LIN {X 0,Y 312.569,Z 301.55,A -85,B 0,C 180,E1 -15776.719,E2 -15776.719} C_VEL
LIN {X 0,Y 312.529,Z 301.553,A -85,B 0,C 180,E1 -15779.646,E2 -15779.646} C_VEL
LIN {X 0,Y 312.5,Z 301.556,A -85,B 0,C 180,E1 -15783.685,E2 -15783.685} C_VEL
LIN {X 0,Y 312.535,Z 301.555,A -85,B 0,C 180,E1 -15787.836,E2 -15787.836} C_VEL
LIN {X 0,Y 312.573,Z 301.686,A -85,B 0,C 180,E1 -15787.985,E2 -15787.985} C_VEL
LIN {X 0,Y 321.169,Z 326.946,A -85,B 0,C 180,E1 -15789.231,E2 -15789.231} C_VEL
LIN {X 0,Y 321.566,Z 328.599,A -85,B 0,C 180,E1 -15789.299,E2 -15789.299} C_VEL
LIN {X 0,Y 319.136,Z 408.879,A -85,B 0,C 180,E1 -15791.461,E2 -15791.461} C_VEL
LIN {X 0,Y 318.645,Z 421.58,A -85,B 0,C 180,E1 -15792.042,E2 -15792.042} C_VEL
LIN {X 0,Y 317.85,Z 434.866,A -85,B 0,C 180,E1 -15792.911,E2 -15792.911} C_VEL
LIN {X 0,Y 316.972,Z 446.153,A -85,B 0,C 180,E1 -15793.897,E2 -15793.897} C_VEL
LIN {X 0,Y 316.011,Z 457.09,A -85,B 0,C 180,E1 -15795.103,E2 -15795.103} C_VEL
LIN {X 0,Y 314.941,Z 468.05,A -85,B 0,C 180,E1 -15796.61,E2 -15796.61} C_VEL
LIN {X 0,Y 313.961,Z 477.57,A -85,B 0,C 180,E1 -15798.246,E2 -15798.246} C_VEL
LIN {X 0,Y 313.106,Z 485.746,A -85,B 0,C 180,E1 -15799.964,E2 -15799.964} C_VEL
LIN {X 0,Y 312.313,Z 493.408,A -85,B 0,C 180,E1 -15801.952,E2 -15801.952} C_VEL
LIN {X 0,Y 311.675,Z 499.881,A -85,B 0,C 180,E1 -15804.108,E2 -15804.108} C_VEL
LIN {X 0,Y 311.305,Z 504.728,A -85,B 0,C 180,E1 -15806.208,E2 -15806.208} C_VEL
LIN {X 0,Y 310.978,Z 507.716,A -85,B 0,C 180,E1 -15807.922,E2 -15807.922} C_VEL
LIN {X 0,Y 310.731,Z 510.421,A -85,B 0,C 180,E1 -15810.16,E2 -15810.16} C_VEL
LIN {X 0,Y 310.726,Z 511.311,A -85,B 0,C 180,E1 -15811.362,E2 -15811.362} C_VEL
LIN {X 0,Y 310.11,Z 511.982,A -85,B 0,C 180,E1 -15812.439,E2 -15812.439} C_VEL
LIN {X 0,Y 307.342,Z 512.482,A -85,B 0,C 180,E1 -15814.207,E2 -15814.207} C_VEL
LIN {X 0,Y 304.699,Z 512.119,A -85,B 0,C 180,E1 -15816.005,E2 -15816.005} C_VEL
LIN {X 0,Y 304.296,Z 511.437,A -85,B 0,C 180,E1 -15817.113,E2 -15817.113} C_VEL
LIN {X 0,Y 304.633,Z 510.361,A -85,B 0,C 180,E1 -15818.339,E2 -15818.339} C_VEL
LIN {X 0,Y 305.421,Z 507.392,A -85,B 0,C 180,E1 -15820.616,E2 -15820.616} C_VEL
LIN {X 0,Y 306.337,Z 503.587,A -85,B 0,C 180,E1 -15822.648,E2 -15822.648} C_VEL
LIN {X 0,Y 307.601,Z 498.313,A -85,B 0,C 180,E1 -15824.767,E2 -15824.767} C_VEL
LIN {X 0,Y 309.165,Z 491.514,A -85,B 0,C 180,E1 -15826.861,E2 -15826.861} C_VEL
LIN {X 0,Y 311.029,Z 482.961,A -85,B 0,C 180,E1 -15828.927,E2 -15828.927} C_VEL
LIN {X 0,Y 312.834,Z 473.936,A -85,B 0,C 180,E1 -15830.66,E2 -15830.66} C_VEL
LIN {X 0,Y 314.861,Z 463.188,A -85,B 0,C 180,E1 -15832.304,E2 -15832.304} C_VEL
LIN {X 0,Y 316.565,Z 452.402,A -85,B 0,C 180,E1 -15833.627,E2 -15833.627} C_VEL
LIN {X 0,Y 318.121,Z 440.675,A -85,B 0,C 180,E1 -15834.752,E2 -15834.752} C_VEL
LIN {X 0,Y 319.445,Z 428.246,A -85,B 0,C 180,E1 -15835.663,E2 -15835.663} C_VEL
LIN {X 0,Y 320.377,Z 416.205,A -85,B 0,C 180,E1 -15836.306,E2 -15836.306} C_VEL
LIN {X 0,Y 321.226,Z 399.512,A -85,B 0,C 180,E1 -15836.865,E2 -15836.865} C_VEL
LIN {X 0,Y 324.423,Z 337.687,A -85,B 0,C 180,E1 -15838.659,E2 -15838.659} C_VEL
LIN {X 0,Y 316.819,Z 321.614,A -85,B 0,C 180,E1 -15840.328,E2 -15840.328} C_VEL
LIN {X 0,Y 311.214,Z 311.88,A -85,B 0,C 180,E1 -15841.598,E2 -15841.598} C_VEL
LIN {X 0,Y 306.346,Z 304.341,A -85,B 0,C 180,E1 -15842.795,E2 -15842.795} C_VEL
LIN {X 0,Y 305.667,Z 302.413,A -85,B 0,C 180,E1 -15843.543,E2 -15843.543} C_VEL
LIN {X 0,Y 305.794,Z 302.393,A -85,B 0,C 180,E1 -15846.599,E2 -15846.599} C_VEL
LIN {X 0,Y 305.658,Z 302.414,A -85,B 0,C 180,E1 -15849.263,E2 -15849.263} C_VEL
LIN {X 0,Y 305.543,Z 302.423,A -85,B 0,C 180,E1 -15853.299,E2 -15853.299} C_VEL
LIN {X 0,Y 305.509,Z 302.428,A -85,B 0,C 180,E1 -15856.025,E2 -15856.025} C_VEL
LIN {X 0,Y 305.442,Z 302.43,A -85,B 0,C 180,E1 -15860.191,E2 -15860.191} C_VEL
LIN {X 0,Y 305.464,Z 302.435,A -85,B 0,C 180,E1 -15864.466,E2 -15864.466} C_VEL
LIN {X 0,Y 305.456,Z 302.438,A -85,B 0,C 180,E1 -15867.398,E2 -15867.398} C_VEL
LIN {X 0,Y 305.402,Z 302.443,A -85,B 0,C 180,E1 -15870.416,E2 -15870.416} C_VEL
LIN {X 0,Y 305.434,Z 302.433,A -85,B 0,C 180,E1 -15874.082,E2 -15874.082} C_VEL
LIN {X 0,Y 305.452,Z 302.432,A -85,B 0,C 180,E1 -15876.743,E2 -15876.743} C_VEL
LIN {X 0,Y 305.435,Z 302.434,A -85,B 0,C 180,E1 -15880.112,E2 -15880.112} C_VEL
LIN {X 0,Y 305.402,Z 302.443,A -85,B 0,C 180,E1 -15883.66,E2 -15883.66} C_VEL
LIN {X 0,Y 305.434,Z 302.44,A -85,B 0,C 180,E1 -15887.419,E2 -15887.419} C_VEL
LIN {X 0,Y 305.457,Z 302.437,A -85,B 0,C 180,E1 -15891.602,E2 -15891.602} C_VEL
LIN {X 0,Y 308.417,Z 311.804,A -85,B 0,C 180,E1 -15895.12,E2 -15895.12} C_VEL
LIN {X 0,Y 311.052,Z 321.561,A -85,B 0,C 180,E1 -15898.326,E2 -15898.326} C_VEL
LIN {X 0,Y 312.487,Z 328.352,A -85,B 0,C 180,E1 -15900.35,E2 -15900.35} C_VEL
LIN {X 0,Y 315.777,Z 336.016,A -85,B 0,C 180,E1 -15901.158,E2 -15901.158} C_VEL
LIN {X 0,Y 319.475,Z 354.495,A -85,B 0,C 180,E1 -15902.374,E2 -15902.374} C_VEL
LIN {X 0,Y 321.978,Z 372.44,A -85,B 0,C 180,E1 -15903.36,E2 -15903.36} C_VEL
LIN {X 0,Y 322.658,Z 381.327,A -85,B 0,C 180,E1 -15903.762,E2 -15903.762} C_VEL
LIN {X 0,Y 319.765,Z 440.74,A -85,B 0,C 180,E1 -15905.495,E2 -15905.495} C_VEL
LIN {X 0,Y 318.351,Z 455.279,A -85,B 0,C 180,E1 -15906.159,E2 -15906.159} C_VEL
LIN {X 0,Y 316.786,Z 467.665,A -85,B 0,C 180,E1 -15906.987,E2 -15906.987} C_VEL
LIN {X 0,Y 314.861,Z 479.761,A -85,B 0,C 180,E1 -15908.05,E2 -15908.05} C_VEL
LIN {X 0,Y 312.782,Z 491.982,A -85,B 0,C 180,E1 -15909.451,E2 -15909.451} C_VEL
LIN {X 0,Y 310.928,Z 501.887,A -85,B 0,C 180,E1 -15910.872,E2 -15910.872} C_VEL
LIN {X 0,Y 309.11,Z 510.986,A -85,B 0,C 180,E1 -15912.471,E2 -15912.471} C_VEL
LIN {X 0,Y 307.444,Z 519.938,A -85,B 0,C 180,E1 -15914.423,E2 -15914.423} C_VEL
LIN {X 0,Y 306.094,Z 527.138,A -85,B 0,C 180,E1 -15916.392,E2 -15916.392} C_VEL
LIN {X 0,Y 305.025,Z 532.101,A -85,B 0,C 180,E1 -15918.035,E2 -15918.035} C_VEL
LIN {X 0,Y 304.335,Z 536.915,A -85,B 0,C 180,E1 -15920.029,E2 -15920.029} C_VEL
LIN {X 0,Y 303.92,Z 540.631,A -85,B 0,C 180,E1 -15922.028,E2 -15922.028} C_VEL
LIN {X 0,Y 303.731,Z 543.552,A -85,B 0,C 180,E1 -15924.257,E2 -15924.257} C_VEL
LIN {X 0,Y 303.708,Z 545.024,A -85,B 0,C 180,E1 -15926.022,E2 -15926.022} C_VEL
LIN {X 0,Y 303.709,Z 545.634,A -85,B 0,C 180,E1 -15927.35,E2 -15927.35} C_VEL
LIN {X 0,Y 303.81,Z 545.808,A -85,B 0,C 180,E1 -15928.677,E2 -15928.677} C_VEL
LIN {X 0,Y 304.002,Z 545.577,A -85,B 0,C 180,E1 -15930.002,E2 -15930.002} C_VEL
LIN {X 0,Y 303.897,Z 544.913,A -85,B 0,C 180,E1 -15931.327,E2 -15931.327} C_VEL
LIN {X 0,Y 303.773,Z 543.775,A -85,B 0,C 180,E1 -15932.654,E2 -15932.654} C_VEL
LIN {X 0,Y 303.805,Z 541.247,A -85,B 0,C 180,E1 -15934.646,E2 -15934.646} C_VEL
LIN {X 0,Y 303.91,Z 537.616,A -85,B 0,C 180,E1 -15936.641,E2 -15936.641} C_VEL
LIN {X 0,Y 304.016,Z 532.776,A -85,B 0,C 180,E1 -15938.643,E2 -15938.643} C_VEL
LIN {X 0,Y 304.449,Z 526.612,A -85,B 0,C 180,E1 -15940.643,E2 -15940.643} C_VEL
LIN {X 0,Y 305.187,Z 518.907,A -85,B 0,C 180,E1 -15942.638,E2 -15942.638} C_VEL
LIN {X 0,Y 305.99,Z 511.012,A -85,B 0,C 180,E1 -15944.295,E2 -15944.295} C_VEL
LIN {X 0,Y 306.916,Z 501.329,A -85,B 0,C 180,E1 -15945.95,E2 -15945.95} C_VEL
LIN {X 0,Y 308.062,Z 490.632,A -85,B 0,C 180,E1 -15947.424,E2 -15947.424} C_VEL
LIN {X 0,Y 309.114,Z 480.385,A -85,B 0,C 180,E1 -15948.561,E2 -15948.561} C_VEL
LIN {X 0,Y 310.224,Z 468.373,A -85,B 0,C 180,E1 -15949.607,E2 -15949.607} C_VEL
LIN {X 0,Y 311.305,Z 454.669,A -85,B 0,C 180,E1 -15950.483,E2 -15950.483} C_VEL
LIN {X 0,Y 312.046,Z 441.896,A -85,B 0,C 180,E1 -15951.036,E2 -15951.036} C_VEL
LIN {X 0,Y 313.768,Z 376.823,A -85,B 0,C 180,E1 -15952.843,E2 -15952.843} C_VEL
LIN {X 0,Y 308.68,Z 334.134,A -85,B 0,C 180,E1 -15954.435,E2 -15954.435} C_VEL
LIN {X 0,Y 309.846,Z 324.126,A -85,B 0,C 180,E1 -15956.977,E2 -15956.977} C_VEL
LIN {X 0,Y 307.598,Z 312.592,A -85,B 0,C 180,E1 -15960.175,E2 -15960.175} C_VEL
LIN {X 0,Y 305.503,Z 302.431,A -85,B 0,C 180,E1 -15963.116,E2 -15963.116} C_VEL
LIN {X 0,Y 305.449,Z 302.439,A -85,B 0,C 180,E1 -15966.741,E2 -15966.741} C_VEL
LIN {X 0,Y 305.403,Z 302.443,A -85,B 0,C 180,E1 -15970.588,E2 -15970.588} C_VEL
LIN {X 0,Y 305.413,Z 302.438,A -85,B 0,C 180,E1 -15973.655,E2 -15973.655} C_VEL
LIN {X 0,Y 305.404,Z 302.44,A -85,B 0,C 180,E1 -15977.421,E2 -15977.421} C_VEL
LIN {X 0,Y 305.417,Z 302.438,A -85,B 0,C 180,E1 -15981.588,E2 -15981.588} C_VEL
LIN {X 0,Y 305.448,Z 302.438,A -85,B 0,C 180,E1 -15984.884,E2 -15984.884} C_VEL
LIN {X 0,Y 305.426,Z 302.437,A -85,B 0,C 180,E1 -15988.358,E2 -15988.358} C_VEL
LIN {X 0,Y 305.473,Z 302.436,A -85,B 0,C 180,E1 -15991.108,E2 -15991.108} C_VEL
LIN {X 0,Y 305.486,Z 302.429,A -85,B 0,C 180,E1 -15994.079,E2 -15994.079} C_VEL
LIN {X 0,Y 305.459,Z 302.436,A -85,B 0,C 180,E1 -15996.974,E2 -15996.974} C_VEL
LIN {X 0,Y 305.498,Z 302.433,A -85,B 0,C 180,E1 -16001.211,E2 -16001.211} C_VEL
LIN {X 0,Y 305.606,Z 302.419,A -85,B 0,C 180,E1 -16005.346,E2 -16005.346} C_VEL
LIN {X 0,Y 305.603,Z 302.42,A -85,B 0,C 180,E1 -16009.398,E2 -16009.398} C_VEL
LIN {X 0,Y 305.765,Z 302.395,A -85,B 0,C 180,E1 -16012.072,E2 -16012.072} C_VEL
LIN {X 0,Y 305.657,Z 302.408,A -85,B 0,C 180,E1 -16014.722,E2 -16014.722} C_VEL
LIN {X 0,Y 305.931,Z 302.374,A -85,B 0,C 180,E1 -16018.683,E2 -16018.683} C_VEL
LIN {X 0,Y 305.931,Z 302.378,A -85,B 0,C 180,E1 -16021.316,E2 -16021.316} C_VEL
LIN {X 0,Y 305.653,Z 302.411,A -85,B 0,C 180,E1 -16025.276,E2 -16025.276} C_VEL
LIN {X 0,Y 305.764,Z 302.397,A -85,B 0,C 180,E1 -16027.926,E2 -16027.926} C_VEL
LIN {X 0,Y 305.58,Z 302.42,A -85,B 0,C 180,E1 -16031.945,E2 -16031.945} C_VEL
LIN {X 0,Y 305.587,Z 302.417,A -85,B 0,C 180,E1 -16035.012,E2 -16035.012} C_VEL
LIN {X 0,Y 305.492,Z 302.428,A -85,B 0,C 180,E1 -16038.788,E2 -16038.788} C_VEL
LIN {X 0,Y 305.469,Z 302.432,A -85,B 0,C 180,E1 -16043.04,E2 -16043.04} C_VEL
LIN {X 0,Y 305.513,Z 302.427,A -85,B 0,C 180,E1 -16046.221,E2 -16046.221} C_VEL
LIN {X 0,Y 305.477,Z 302.43,A -85,B 0,C 180,E1 -16049.05,E2 -16049.05} C_VEL
LIN {X 0,Y 305.428,Z 302.441,A -85,B 0,C 180,E1 -16051.953,E2 -16051.953} C_VEL
LIN {X 0,Y 305.446,Z 302.434,A -85,B 0,C 180,E1 -16055.114,E2 -16055.114} C_VEL
LIN {X 0,Y 305.454,Z 302.434,A -85,B 0,C 180,E1 -16058.534,E2 -16058.534} C_VEL
LIN {X 0,Y 305.449,Z 302.434,A -85,B 0,C 180,E1 -16062.588,E2 -16062.588} C_VEL
LIN {X 0,Y 305.476,Z 302.433,A -85,B 0,C 180,E1 -16066.357,E2 -16066.357} C_VEL
LIN {X 0,Y 305.475,Z 302.434,A -85,B 0,C 180,E1 -16069.897,E2 -16069.897} C_VEL
LIN {X 0,Y 305.494,Z 302.429,A -85,B 0,C 180,E1 -16073.627,E2 -16073.627} C_VEL
LIN {X 0,Y 305.458,Z 302.436,A -85,B 0,C 180,E1 -16076.484,E2 -16076.484} C_VEL
LIN {X 0,Y 305.451,Z 302.434,A -85,B 0,C 180,E1 -16079.591,E2 -16079.591} C_VEL
LIN {X 0,Y 305.513,Z 302.428,A -85,B 0,C 180,E1 -16082.608,E2 -16082.608} C_VEL
LIN {X 0,Y 305.504,Z 302.427,A -85,B 0,C 180,E1 -16085.539,E2 -16085.539} C_VEL
LIN {X 0,Y 305.516,Z 302.426,A -85,B 0,C 180,E1 -16089.815,E2 -16089.815} C_VEL
LIN {X 0,Y 305.572,Z 302.422,A -85,B 0,C 180,E1 -16092.602,E2 -16092.602} C_VEL
LIN {X 0,Y 305.646,Z 302.409,A -85,B 0,C 180,E1 -16095.348,E2 -16095.348} C_VEL
LIN {X 0,Y 305.636,Z 302.41,A -85,B 0,C 180,E1 -16099.399,E2 -16099.399} C_VEL
LIN {X 0,Y 305.811,Z 302.39,A -85,B 0,C 180,E1 -16102.073,E2 -16102.073} C_VEL
LIN {X 0,Y 305.686,Z 302.408,A -85,B 0,C 180,E1 -16104.722,E2 -16104.722} C_VEL
LIN {X 0,Y 305.955,Z 302.376,A -85,B 0,C 180,E1 -16108.682,E2 -16108.682} C_VEL
LIN {X 0,Y 305.954,Z 302.371,A -85,B 0,C 180,E1 -16111.314,E2 -16111.314} C_VEL
LIN {X 0,Y 305.846,Z 302.388,A -85,B 0,C 180,E1 -16116.595,E2 -16116.595} C_VEL
LIN {X 0,Y 305.73,Z 302.4,A -85,B 0,C 180,E1 -16119.257,E2 -16119.257} C_VEL
LIN {X 0,Y 305.584,Z 302.419,A -85,B 0,C 180,E1 -16123.293,E2 -16123.293} C_VEL
LIN {X 0,Y 305.585,Z 302.416,A -85,B 0,C 180,E1 -16126.017,E2 -16126.017} C_VEL
LIN {X 0,Y 305.603,Z 302.416,A -85,B 0,C 180,E1 -16129.461,E2 -16129.461} C_VEL
LIN {X 0,Y 305.481,Z 302.435,A -85,B 0,C 180,E1 -16133.039,E2 -16133.039} C_VEL
LIN {X 0,Y 305.54,Z 302.423,A -85,B 0,C 180,E1 -16136.226,E2 -16136.226} C_VEL
LIN {X 0,Y 305.48,Z 302.436,A -85,B 0,C 180,E1 -16139.046,E2 -16139.046} C_VEL
LIN {X 0,Y 305.446,Z 302.436,A -85,B 0,C 180,E1 -16143.513,E2 -16143.513} C_VEL
LIN {X 0,Y 305.504,Z 302.431,A -85,B 0,C 180,E1 -16147.555,E2 -16147.555} C_VEL
LIN {X 0,Y 312.503,Z 322.639,A -85,B 0,C 180,E1 -16148.602,E2 -16148.602} C_VEL
LIN {X 0,Y 314.751,Z 329.425,A -85,B 0,C 180,E1 -16148.934,E2 -16148.934} C_VEL
LIN {X 0,Y 312.289,Z 408.997,A -85,B 0,C 180,E1 -16151.132,E2 -16151.132} C_VEL
LIN {X 0,Y 311.764,Z 421.741,A -85,B 0,C 180,E1 -16151.724,E2 -16151.724} C_VEL
LIN {X 0,Y 310.939,Z 435.162,A -85,B 0,C 180,E1 -16152.617,E2 -16152.617} C_VEL
LIN {X 0,Y 309.981,Z 447.296,A -85,B 0,C 180,E1 -16153.712,E2 -16153.712} C_VEL
LIN {X 0,Y 309,Z 457.772,A -85,B 0,C 180,E1 -16154.904,E2 -16154.904} C_VEL
LIN {X 0,Y 307.983,Z 468.06,A -85,B 0,C 180,E1 -16156.348,E2 -16156.348} C_VEL
LIN {X 0,Y 306.9,Z 478.402,A -85,B 0,C 180,E1 -16158.168,E2 -16158.168} C_VEL
LIN {X 0,Y 305.951,Z 486.707,A -85,B 0,C 180,E1 -16159.971,E2 -16159.971} C_VEL
LIN {X 0,Y 305.193,Z 494.139,A -85,B 0,C 180,E1 -16161.976,E2 -16161.976} C_VEL
LIN {X 0,Y 304.535,Z 500.825,A -85,B 0,C 180,E1 -16164.292,E2 -16164.292} C_VEL
LIN {X 0,Y 304.192,Z 505.321,A -85,B 0,C 180,E1 -16166.325,E2 -16166.325} C_VEL
LIN {X 0,Y 303.76,Z 509.324,A -85,B 0,C 180,E1 -16168.863,E2 -16168.863} C_VEL
LIN {X 0,Y 303.669,Z 511.812,A -85,B 0,C 180,E1 -16171.562,E2 -16171.562} C_VEL
LIN {X 0,Y 303.821,Z 512.519,A -85,B 0,C 180,E1 -16174.425,E2 -16174.425} C_VEL
LIN {X 0,Y 304.296,Z 511.437,A -85,B 0,C 180,E1 -16177.113,E2 -16177.113} C_VEL
LIN {X 0,Y 303.951,Z 510.564,A -85,B 0,C 180,E1 -16178.21,E2 -16178.21} C_VEL
LIN {X 0,Y 301.661,Z 508.799,A -85,B 0,C 180,E1 -16180.007,E2 -16180.007} C_VEL
LIN {X 0,Y 299.514,Z 506.398,A -85,B 0,C 180,E1 -16181.799,E2 -16181.799} C_VEL
LIN {X 0,Y 299.401,Z 504.432,A -85,B 0,C 180,E1 -16182.871,E2 -16182.871} C_VEL
LIN {X 0,Y 300.781,Z 499.083,A -85,B 0,C 180,E1 -16185.107,E2 -16185.107} C_VEL
LIN {X 0,Y 302.515,Z 492.13,A -85,B 0,C 180,E1 -16187.318,E2 -16187.318} C_VEL
LIN {X 0,Y 304.408,Z 483.974,A -85,B 0,C 180,E1 -16189.357,E2 -16189.357} C_VEL
LIN {X 0,Y 306.286,Z 475.271,A -85,B 0,C 180,E1 -16191.102,E2 -16191.102} C_VEL
LIN {X 0,Y 308.234,Z 465.715,A -85,B 0,C 180,E1 -16192.632,E2 -16192.632} C_VEL
LIN {X 0,Y 309.994,Z 455.269,A -85,B 0,C 180,E1 -16193.993,E2 -16193.993} C_VEL
LIN {X 0,Y 311.672,Z 444.087,A -85,B 0,C 180,E1 -16195.15,E2 -16195.15} C_VEL
LIN {X 0,Y 313.129,Z 431.723,A -85,B 0,C 180,E1 -16196.14,E2 -16196.14} C_VEL
LIN {X 0,Y 314.275,Z 419.181,A -85,B 0,C 180,E1 -16196.876,E2 -16196.876} C_VEL
LIN {X 0,Y 315.039,Z 406.996,A -85,B 0,C 180,E1 -16197.363,E2 -16197.363} C_VEL
LIN {X 0,Y 318.65,Z 339.96,A -85,B 0,C 180,E1 -16199.357,E2 -16199.357} C_VEL
LIN {X 0,Y 311.717,Z 325.283,A -85,B 0,C 180,E1 -16200.971,E2 -16200.971} C_VEL
LIN {X 0,Y 306.646,Z 316.358,A -85,B 0,C 180,E1 -16202.174,E2 -16202.174} C_VEL
LIN {X 0,Y 301.652,Z 308.919,A -85,B 0,C 180,E1 -16203.407,E2 -16203.407} C_VEL
LIN {X 0,Y 299.041,Z 305.144,A -85,B 0,C 180,E1 -16204.128,E2 -16204.128} C_VEL
LIN {X 0,Y 298.594,Z 303.291,A -85,B 0,C 180,E1 -16204.895,E2 -16204.895} C_VEL
LIN {X 0,Y 298.739,Z 303.273,A -85,B 0,C 180,E1 -16206.756,E2 -16206.756} C_VEL
LIN {X 0,Y 298.59,Z 303.293,A -85,B 0,C 180,E1 -16209.484,E2 -16209.484} C_VEL
LIN {X 0,Y 298.503,Z 303.303,A -85,B 0,C 180,E1 -16213.618,E2 -16213.618} C_VEL
LIN {X 0,Y 298.442,Z 303.31,A -85,B 0,C 180,E1 -16216.415,E2 -16216.415} C_VEL
LIN {X 0,Y 298.405,Z 303.31,A -85,B 0,C 180,E1 -16219.62,E2 -16219.62} C_VEL
LIN {X 0,Y 298.392,Z 303.311,A -85,B 0,C 180,E1 -16223.604,E2 -16223.604} C_VEL
LIN {X 0,Y 298.425,Z 303.307,A -85,B 0,C 180,E1 -16226.581,E2 -16226.581} C_VEL
LIN {X 0,Y 298.37,Z 303.316,A -85,B 0,C 180,E1 -16229.647,E2 -16229.647} C_VEL
LIN {X 0,Y 298.361,Z 303.318,A -85,B 0,C 180,E1 -16232.805,E2 -16232.805} C_VEL
LIN {X 0,Y 298.423,Z 303.307,A -85,B 0,C 180,E1 -16236.813,E2 -16236.813} C_VEL
LIN {X 0,Y 298.389,Z 303.312,A -85,B 0,C 180,E1 -16239.49,E2 -16239.49} C_VEL
LIN {X 0,Y 298.377,Z 303.317,A -85,B 0,C 180,E1 -16243.108,E2 -16243.108} C_VEL
LIN {X 0,Y 298.383,Z 303.315,A -85,B 0,C 180,E1 -16246.926,E2 -16246.926} C_VEL
LIN {X 0,Y 298.404,Z 303.446,A -85,B 0,C 180,E1 -16250.411,E2 -16250.411} C_VEL
LIN {X 0,Y 301.282,Z 312.125,A -85,B 0,C 180,E1 -16253.897,E2 -16253.897} C_VEL
LIN {X 0,Y 303.981,Z 321.75,A -85,B 0,C 180,E1 -16257.276,E2 -16257.276} C_VEL
LIN {X 0,Y 305.376,Z 327.791,A -85,B 0,C 180,E1 -16259.165,E2 -16259.165} C_VEL
LIN {X 0,Y 310.513,Z 339.127,A -85,B 0,C 180,E1 -16260.474,E2 -16260.474} C_VEL
LIN {X 0,Y 313.87,Z 356.502,A -85,B 0,C 180,E1 -16261.673,E2 -16261.673} C_VEL
LIN {X 0,Y 316.164,Z 373.165,A -85,B 0,C 180,E1 -16262.621,E2 -16262.621} C_VEL
LIN {X 0,Y 316.888,Z 381.023,A -85,B 0,C 180,E1 -16263.009,E2 -16263.009} C_VEL
LIN {X 0,Y 313.739,Z 440.814,A -85,B 0,C 180,E1 -16264.815,E2 -16264.815} C_VEL
LIN {X 0,Y 312.283,Z 455.163,A -85,B 0,C 180,E1 -16265.489,E2 -16265.489} C_VEL
LIN {X 0,Y 310.635,Z 467.444,A -85,B 0,C 180,E1 -16266.327,E2 -16266.327} C_VEL
LIN {X 0,Y 308.613,Z 479.502,A -85,B 0,C 180,E1 -16267.405,E2 -16267.405} C_VEL
LIN {X 0,Y 306.688,Z 490.483,A -85,B 0,C 180,E1 -16268.672,E2 -16268.672} C_VEL
LIN {X 0,Y 304.659,Z 500.524,A -85,B 0,C 180,E1 -16270.112,E2 -16270.112} C_VEL
LIN {X 0,Y 302.725,Z 509.719,A -85,B 0,C 180,E1 -16271.739,E2 -16271.739} C_VEL
LIN {X 0,Y 300.818,Z 518.805,A -85,B 0,C 180,E1 -16273.723,E2 -16273.723} C_VEL
LIN {X 0,Y 299.389,Z 526.169,A -85,B 0,C 180,E1 -16275.734,E2 -16275.734} C_VEL
LIN {X 0,Y 298.049,Z 532.096,A -85,B 0,C 180,E1 -16277.751,E2 -16277.751} C_VEL
LIN {X 0,Y 297.323,Z 536.809,A -85,B 0,C 180,E1 -16279.792,E2 -16279.792} C_VEL
LIN {X 0,Y 296.858,Z 540.427,A -85,B 0,C 180,E1 -16281.837,E2 -16281.837} C_VEL
LIN {X 0,Y 296.601,Z 543.687,A -85,B 0,C 180,E1 -16284.564,E2 -16284.564} C_VEL
LIN {X 0,Y 296.62,Z 544.695,A -85,B 0,C 180,E1 -16285.927,E2 -16285.927} C_VEL
LIN {X 0,Y 296.63,Z 545.239,A -85,B 0,C 180,E1 -16287.286,E2 -16287.286} C_VEL
LIN {X 0,Y 296.717,Z 545.375,A -85,B 0,C 180,E1 -16288.645,E2 -16288.645} C_VEL
LIN {X 0,Y 296.927,Z 545.108,A -85,B 0,C 180,E1 -16290.002,E2 -16290.002} C_VEL
LIN {X 0,Y 296.806,Z 544.383,A -85,B 0,C 180,E1 -16291.359,E2 -16291.359} C_VEL
LIN {X 0,Y 296.693,Z 543.183,A -85,B 0,C 180,E1 -16292.717,E2 -16292.717} C_VEL
LIN {X 0,Y 296.732,Z 540.567,A -85,B 0,C 180,E1 -16294.757,E2 -16294.757} C_VEL
LIN {X 0,Y 296.84,Z 536.847,A -85,B 0,C 180,E1 -16296.8,E2 -16296.8} C_VEL
LIN {X 0,Y 296.965,Z 531.91,A -85,B 0,C 180,E1 -16298.85,E2 -16298.85} C_VEL
LIN {X 0,Y 297.42,Z 525.64,A -85,B 0,C 180,E1 -16300.898,E2 -16300.898} C_VEL
LIN {X 0,Y 298.193,Z 517.798,A -85,B 0,C 180,E1 -16302.939,E2 -16302.939} C_VEL
LIN {X 0,Y 299.084,Z 509.731,A -85,B 0,C 180,E1 -16304.633,E2 -16304.633} C_VEL
LIN {X 0,Y 300.055,Z 499.854,A -85,B 0,C 180,E1 -16306.325,E2 -16306.325} C_VEL
LIN {X 0,Y 301.271,Z 488.949,A -85,B 0,C 180,E1 -16307.829,E2 -16307.829} C_VEL
LIN {X 0,Y 302.563,Z 476.631,A -85,B 0,C 180,E1 -16309.154,E2 -16309.154} C_VEL
LIN {X 0,Y 303.669,Z 464.764,A -85,B 0,C 180,E1 -16310.137,E2 -16310.137} C_VEL
LIN {X 0,Y 304.563,Z 452.075,A -85,B 0,C 180,E1 -16310.913,E2 -16310.913} C_VEL
LIN {X 0,Y 305.266,Z 439.188,A -85,B 0,C 180,E1 -16311.437,E2 -16311.437} C_VEL
LIN {X 0,Y 306.954,Z 377.521,A -85,B 0,C 180,E1 -16313.197,E2 -16313.197} C_VEL
LIN {X 0,Y 301.816,Z 333.82,A -85,B 0,C 180,E1 -16314.854,E2 -16314.854} C_VEL
LIN {X 0,Y 302.819,Z 325.9,A -85,B 0,C 180,E1 -16316.908,E2 -16316.908} C_VEL
LIN {X 0,Y 301.341,Z 317.262,A -85,B 0,C 180,E1 -16319.325,E2 -16319.325} C_VEL
LIN {X 0,Y 298.446,Z 303.309,A -85,B 0,C 180,E1 -16323.422,E2 -16323.422} C_VEL
LIN {X 0,Y 298.385,Z 303.313,A -85,B 0,C 180,E1 -16327.761,E2 -16327.761} C_VEL
LIN {X 0,Y 298.341,Z 303.321,A -85,B 0,C 180,E1 -16331.267,E2 -16331.267} C_VEL
LIN {X 0,Y 298.349,Z 303.322,A -85,B 0,C 180,E1 -16335.033,E2 -16335.033} C_VEL
LIN {X 0,Y 298.332,Z 303.326,A -85,B 0,C 180,E1 -16338.921,E2 -16338.921} C_VEL
LIN {X 0,Y 298.367,Z 303.316,A -85,B 0,C 180,E1 -16342.234,E2 -16342.234} C_VEL
LIN {X 0,Y 298.395,Z 303.314,A -85,B 0,C 180,E1 -16345.579,E2 -16345.579} C_VEL
LIN {X 0,Y 298.362,Z 303.32,A -85,B 0,C 180,E1 -16348.787,E2 -16348.787} C_VEL
LIN {X 0,Y 298.409,Z 303.311,A -85,B 0,C 180,E1 -16351.898,E2 -16351.898} C_VEL
LIN {X 0,Y 298.424,Z 303.312,A -85,B 0,C 180,E1 -16354.918,E2 -16354.918} C_VEL
LIN {X 0,Y 298.382,Z 303.314,A -85,B 0,C 180,E1 -16357.86,E2 -16357.86} C_VEL
LIN {X 0,Y 298.445,Z 303.308,A -85,B 0,C 180,E1 -16360.75,E2 -16360.75} C_VEL
LIN {X 0,Y 298.57,Z 303.293,A -85,B 0,C 180,E1 -16364.993,E2 -16364.993} C_VEL
LIN {X 0,Y 298.562,Z 303.295,A -85,B 0,C 180,E1 -16369.145,E2 -16369.145} C_VEL
LIN {X 0,Y 298.711,Z 303.274,A -85,B 0,C 180,E1 -16371.884,E2 -16371.884} C_VEL
LIN {X 0,Y 298.628,Z 303.283,A -85,B 0,C 180,E1 -16374.598,E2 -16374.598} C_VEL
LIN {X 0,Y 298.898,Z 303.25,A -85,B 0,C 180,E1 -16378.652,E2 -16378.652} C_VEL
LIN {X 0,Y 298.897,Z 303.254,A -85,B 0,C 180,E1 -16381.347,E2 -16381.347} C_VEL
LIN {X 0,Y 298.75,Z 303.268,A -85,B 0,C 180,E1 -16386.754,E2 -16386.754} C_VEL
LIN {X 0,Y 298.611,Z 303.29,A -85,B 0,C 180,E1 -16389.482,E2 -16389.482} C_VEL
LIN {X 0,Y 298.522,Z 303.302,A -85,B 0,C 180,E1 -16393.616,E2 -16393.616} C_VEL
LIN {X 0,Y 298.458,Z 303.305,A -85,B 0,C 180,E1 -16396.413,E2 -16396.413} C_VEL
LIN {X 0,Y 298.423,Z 303.313,A -85,B 0,C 180,E1 -16399.617,E2 -16399.617} C_VEL
LIN {X 0,Y 298.411,Z 303.314,A -85,B 0,C 180,E1 -16403.601,E2 -16403.601} C_VEL
LIN {X 0,Y 298.471,Z 303.303,A -85,B 0,C 180,E1 -16406.575,E2 -16406.575} C_VEL
LIN {X 0,Y 298.404,Z 303.315,A -85,B 0,C 180,E1 -16409.642,E2 -16409.642} C_VEL
LIN {X 0,Y 298.38,Z 303.314,A -85,B 0,C 180,E1 -16412.801,E2 -16412.801} C_VEL
LIN {X 0,Y 298.432,Z 303.307,A -85,B 0,C 180,E1 -16416.808,E2 -16416.808} C_VEL
LIN {X 0,Y 298.397,Z 303.314,A -85,B 0,C 180,E1 -16419.487,E2 -16419.487} C_VEL
LIN {X 0,Y 298.388,Z 303.313,A -85,B 0,C 180,E1 -16423.104,E2 -16423.104} C_VEL
LIN {X 0,Y 298.429,Z 303.308,A -85,B 0,C 180,E1 -16426.928,E2 -16426.928} C_VEL
LIN {X 0,Y 298.421,Z 303.311,A -85,B 0,C 180,E1 -16430.518,E2 -16430.518} C_VEL
LIN {X 0,Y 298.426,Z 303.311,A -85,B 0,C 180,E1 -16433.933,E2 -16433.933} C_VEL
LIN {X 0,Y 298.387,Z 303.317,A -85,B 0,C 180,E1 -16437.985,E2 -16437.985} C_VEL
LIN {X 0,Y 298.453,Z 303.307,A -85,B 0,C 180,E1 -16441.904,E2 -16441.904} C_VEL
LIN {X 0,Y 298.481,Z 303.303,A -85,B 0,C 180,E1 -16444.924,E2 -16444.924} C_VEL
LIN {X 0,Y 298.455,Z 303.304,A -85,B 0,C 180,E1 -16449.316,E2 -16449.316} C_VEL
LIN {X 0,Y 298.535,Z 303.298,A -85,B 0,C 180,E1 -16452.179,E2 -16452.179} C_VEL
LIN {X 0,Y 298.591,Z 303.289,A -85,B 0,C 180,E1 -16454.994,E2 -16454.994} C_VEL
LIN {X 0,Y 298.591,Z 303.288,A -85,B 0,C 180,E1 -16459.145,E2 -16459.145} C_VEL
LIN {X 0,Y 298.756,Z 303.268,A -85,B 0,C 180,E1 -16461.885,E2 -16461.885} C_VEL
LIN {X 0,Y 298.658,Z 303.285,A -85,B 0,C 180,E1 -16464.597,E2 -16464.597} C_VEL
LIN {X 0,Y 298.921,Z 303.252,A -85,B 0,C 180,E1 -16468.651,E2 -16468.651} C_VEL
LIN {X 0,Y 298.921,Z 303.247,A -85,B 0,C 180,E1 -16471.345,E2 -16471.345} C_VEL
LIN {X 0,Y 298.792,Z 303.269,A -85,B 0,C 180,E1 -16476.751,E2 -16476.751} C_VEL
LIN {X 0,Y 298.675,Z 303.278,A -85,B 0,C 180,E1 -16479.477,E2 -16479.477} C_VEL
LIN {X 0,Y 298.546,Z 303.294,A -85,B 0,C 180,E1 -16483.612,E2 -16483.612} C_VEL
LIN {X 0,Y 298.541,Z 303.296,A -85,B 0,C 180,E1 -16486.405,E2 -16486.405} C_VEL
LIN {X 0,Y 298.532,Z 303.296,A -85,B 0,C 180,E1 -16489.667,E2 -16489.667} C_VEL
LIN {X 0,Y 298.447,Z 303.307,A -85,B 0,C 180,E1 -16493.594,E2 -16493.594} C_VEL
LIN {X 0,Y 298.478,Z 303.304,A -85,B 0,C 180,E1 -16496.57,E2 -16496.57} C_VEL
LIN {X 0,Y 298.405,Z 303.312,A -85,B 0,C 180,E1 -16499.637,E2 -16499.637} C_VEL
LIN {X 0,Y 298.377,Z 303.318,A -85,B 0,C 180,E1 -16502.796,E2 -16502.796} C_VEL
LIN {X 0,Y 298.446,Z 303.311,A -85,B 0,C 180,E1 -16506.927,E2 -16506.927} C_VEL
LIN {X 0,Y 298.439,Z 303.312,A -85,B 0,C 180,E1 -16507.145,E2 -16507.145} C_VEL
LIN {X 0,Y 305.918,Z 324.639,A -85,B 0,C 180,E1 -16508.277,E2 -16508.277} C_VEL
LIN {X 0,Y 307.933,Z 330.728,A -85,B 0,C 180,E1 -16508.579,E2 -16508.579} C_VEL
LIN {X 0,Y 305.415,Z 409.265,A -85,B 0,C 180,E1 -16510.814,E2 -16510.814} C_VEL
LIN {X 0,Y 304.877,Z 422.037,A -85,B 0,C 180,E1 -16511.421,E2 -16511.421} C_VEL
LIN {X 0,Y 304.067,Z 435.063,A -85,B 0,C 180,E1 -16512.302,E2 -16512.302} C_VEL
LIN {X 0,Y 303.138,Z 446.464,A -85,B 0,C 180,E1 -16513.332,E2 -16513.332} C_VEL
LIN {X 0,Y 301.939,Z 458.909,A -85,B 0,C 180,E1 -16514.772,E2 -16514.772} C_VEL
LIN {X 0,Y 300.87,Z 469.844,A -85,B 0,C 180,E1 -16516.387,E2 -16516.387} C_VEL
LIN {X 0,Y 299.76,Z 479.778,A -85,B 0,C 180,E1 -16518.211,E2 -16518.211} C_VEL
LIN {X 0,Y 298.786,Z 488.221,A -85,B 0,C 180,E1 -16520.137,E2 -16520.137} C_VEL
LIN {X 0,Y 298.033,Z 495.399,A -85,B 0,C 180,E1 -16522.186,E2 -16522.186} C_VEL
LIN {X 0,Y 297.477,Z 501.079,A -85,B 0,C 180,E1 -16524.217,E2 -16524.217} C_VEL
LIN {X 0,Y 297.071,Z 505.893,A -85,B 0,C 180,E1 -16526.439,E2 -16526.439} C_VEL
LIN {X 0,Y 296.697,Z 509.305,A -85,B 0,C 180,E1 -16528.593,E2 -16528.593} C_VEL
LIN {X 0,Y 296.573,Z 511.914,A -85,B 0,C 180,E1 -16531.244,E2 -16531.244} C_VEL
LIN {X 0,Y 296.591,Z 512.84,A -85,B 0,C 180,E1 -16533.243,E2 -16533.243} C_VEL
LIN {X 0,Y 296.788,Z 512.939,A -85,B 0,C 180,E1 -16534.771,E2 -16534.771} C_VEL
LIN {X 0,Y 297.241,Z 512.014,A -85,B 0,C 180,E1 -16537.219,E2 -16537.219} C_VEL
LIN {X 0,Y 297.875,Z 510.167,A -85,B 0,C 180,E1 -16539.274,E2 -16539.274} C_VEL
LIN {X 0,Y 298.714,Z 507.058,A -85,B 0,C 180,E1 -16541.482,E2 -16541.482} C_VEL
LIN {X 0,Y 299.401,Z 504.432,A -85,B 0,C 180,E1 -16542.871,E2 -16542.871} C_VEL
LIN {X 0,Y 299.374,Z 502.291,A -85,B 0,C 180,E1 -16543.924,E2 -16543.924} C_VEL
LIN {X 0,Y 297.704,Z 498.521,A -85,B 0,C 180,E1 -16545.655,E2 -16545.655} C_VEL
LIN {X 0,Y 296.163,Z 494.144,A -85,B 0,C 180,E1 -16547.344,E2 -16547.344} C_VEL
LIN {X 0,Y 296.331,Z 491.002,A -85,B 0,C 180,E1 -16548.313,E2 -16548.313} C_VEL
LIN {X 0,Y 298.181,Z 483.485,A -85,B 0,C 180,E1 -16550.162,E2 -16550.162} C_VEL
LIN {X 0,Y 300.213,Z 474.543,A -85,B 0,C 180,E1 -16551.926,E2 -16551.926} C_VEL
LIN {X 0,Y 302.567,Z 463.247,A -85,B 0,C 180,E1 -16553.7,E2 -16553.7} C_VEL
LIN {X 0,Y 304.416,Z 452.575,A -85,B 0,C 180,E1 -16555.034,E2 -16555.034} C_VEL
LIN {X 0,Y 306.329,Z 439.52,A -85,B 0,C 180,E1 -16556.301,E2 -16556.301} C_VEL
LIN {X 0,Y 307.8,Z 426.69,A -85,B 0,C 180,E1 -16557.22,E2 -16557.22} C_VEL
LIN {X 0,Y 308.839,Z 413.612,A -85,B 0,C 180,E1 -16557.885,E2 -16557.885} C_VEL
LIN {X 0,Y 312.958,Z 342.452,A -85,B 0,C 180,E1 -16560.084,E2 -16560.084} C_VEL
LIN {X 0,Y 307.145,Z 329.862,A -85,B 0,C 180,E1 -16561.515,E2 -16561.515} C_VEL
LIN {X 0,Y 302.402,Z 321.304,A -85,B 0,C 180,E1 -16562.715,E2 -16562.715} C_VEL
LIN {X 0,Y 297.658,Z 314.108,A -85,B 0,C 180,E1 -16563.935,E2 -16563.935} C_VEL
LIN {X 0,Y 292.067,Z 306.004,A -85,B 0,C 180,E1 -16565.524,E2 -16565.524} C_VEL
LIN {X 0,Y 291.666,Z 304.153,A -85,B 0,C 180,E1 -16566.399,E2 -16566.399} C_VEL
LIN {X 0,Y 291.532,Z 304.17,A -85,B 0,C 180,E1 -16569.716,E2 -16569.716} C_VEL
LIN {X 0,Y 291.474,Z 304.179,A -85,B 0,C 180,E1 -16573.953,E2 -16573.953} C_VEL
LIN {X 0,Y 291.387,Z 304.186,A -85,B 0,C 180,E1 -16576.824,E2 -16576.824} C_VEL
LIN {X 0,Y 291.355,Z 304.186,A -85,B 0,C 180,E1 -16579.845,E2 -16579.845} C_VEL
LIN {X 0,Y 291.343,Z 304.193,A -85,B 0,C 180,E1 -16584.211,E2 -16584.211} C_VEL
LIN {X 0,Y 291.368,Z 304.192,A -85,B 0,C 180,E1 -16587.278,E2 -16587.278} C_VEL
LIN {X 0,Y 291.29,Z 304.202,A -85,B 0,C 180,E1 -16590.443,E2 -16590.443} C_VEL
LIN {X 0,Y 291.313,Z 304.194,A -85,B 0,C 180,E1 -16593.703,E2 -16593.703} C_VEL
LIN {X 0,Y 291.36,Z 304.186,A -85,B 0,C 180,E1 -16597.261,E2 -16597.261} C_VEL
LIN {X 0,Y 291.313,Z 304.197,A -85,B 0,C 180,E1 -16600.647,E2 -16600.647} C_VEL
LIN {X 0,Y 291.269,Z 304.2,A -85,B 0,C 180,E1 -16604.407,E2 -16604.407} C_VEL
LIN {X 0,Y 291.309,Z 304.197,A -85,B 0,C 180,E1 -16608.59,E2 -16608.59} C_VEL
LIN {X 0,Y 291.357,Z 304.341,A -85,B 0,C 180,E1 -16608.985,E2 -16608.985} C_VEL
LIN {X 0,Y 293.774,Z 311.494,A -85,B 0,C 180,E1 -16612.136,E2 -16612.136} C_VEL
LIN {X 0,Y 295.992,Z 318.576,A -85,B 0,C 180,E1 -16614.914,E2 -16614.914} C_VEL
LIN {X 0,Y 298.169,Z 326.91,A -85,B 0,C 180,E1 -16617.823,E2 -16617.823} C_VEL
LIN {X 0,Y 303.773,Z 338.761,A -85,B 0,C 180,E1 -16619.364,E2 -16619.364} C_VEL
LIN {X 0,Y 305.611,Z 343.284,A -85,B 0,C 180,E1 -16619.862,E2 -16619.862} C_VEL
LIN {X 0,Y 308.841,Z 361.489,A -85,B 0,C 180,E1 -16621.122,E2 -16621.122} C_VEL
LIN {X 0,Y 310.887,Z 378.75,A -85,B 0,C 180,E1 -16622.107,E2 -16622.107} C_VEL
LIN {X 0,Y 311.076,Z 383.685,A -85,B 0,C 180,E1 -16622.323,E2 -16622.323} C_VEL
LIN {X 0,Y 307.95,Z 439.704,A -85,B 0,C 180,E1 -16624.04,E2 -16624.04} C_VEL
LIN {X 0,Y 306.473,Z 454.008,A -85,B 0,C 180,E1 -16624.721,E2 -16624.721} C_VEL
LIN {X 0,Y 304.849,Z 465.454,A -85,B 0,C 180,E1 -16625.487,E2 -16625.487} C_VEL
LIN {X 0,Y 302.721,Z 477.723,A -85,B 0,C 180,E1 -16626.578,E2 -16626.578} C_VEL
LIN {X 0,Y 300.372,Z 490.193,A -85,B 0,C 180,E1 -16628.02,E2 -16628.02} C_VEL
LIN {X 0,Y 298.033,Z 501.195,A -85,B 0,C 180,E1 -16629.65,E2 -16629.65} C_VEL
LIN {X 0,Y 296.005,Z 510.224,A -85,B 0,C 180,E1 -16631.309,E2 -16631.309} C_VEL
LIN {X 0,Y 294.015,Z 519.114,A -85,B 0,C 180,E1 -16633.335,E2 -16633.335} C_VEL
LIN {X 0,Y 292.503,Z 526.273,A -85,B 0,C 180,E1 -16635.391,E2 -16635.391} C_VEL
LIN {X 0,Y 291.088,Z 532.092,A -85,B 0,C 180,E1 -16637.453,E2 -16637.453} C_VEL
LIN {X 0,Y 290.303,Z 536.713,A -85,B 0,C 180,E1 -16639.542,E2 -16639.542} C_VEL
LIN {X 0,Y 289.816,Z 540.245,A -85,B 0,C 180,E1 -16641.637,E2 -16641.637} C_VEL
LIN {X 0,Y 289.537,Z 543.418,A -85,B 0,C 180,E1 -16644.431,E2 -16644.431} C_VEL
LIN {X 0,Y 289.534,Z 544.343,A -85,B 0,C 180,E1 -16645.827,E2 -16645.827} C_VEL
LIN {X 0,Y 289.552,Z 544.847,A -85,B 0,C 180,E1 -16647.22,E2 -16647.22} C_VEL
LIN {X 0,Y 289.624,Z 544.945,A -85,B 0,C 180,E1 -16648.612,E2 -16648.612} C_VEL
LIN {X 0,Y 289.838,Z 544.636,A -85,B 0,C 180,E1 -16650.002,E2 -16650.002} C_VEL
LIN {X 0,Y 289.715,Z 543.833,A -85,B 0,C 180,E1 -16651.392,E2 -16651.392} C_VEL
LIN {X 0,Y 289.617,Z 542.592,A -85,B 0,C 180,E1 -16652.784,E2 -16652.784} C_VEL
LIN {X 0,Y 289.664,Z 539.887,A -85,B 0,C 180,E1 -16654.873,E2 -16654.873} C_VEL
LIN {X 0,Y 289.749,Z 536.068,A -85,B 0,C 180,E1 -16656.967,E2 -16656.967} C_VEL
LIN {X 0,Y 289.925,Z 531.029,A -85,B 0,C 180,E1 -16659.067,E2 -16659.067} C_VEL
LIN {X 0,Y 290.376,Z 524.635,A -85,B 0,C 180,E1 -16661.166,E2 -16661.166} C_VEL
LIN {X 0,Y 291.228,Z 516.601,A -85,B 0,C 180,E1 -16663.254,E2 -16663.254} C_VEL
LIN {X 0,Y 292.176,Z 508.372,A -85,B 0,C 180,E1 -16664.987,E2 -16664.987} C_VEL
LIN {X 0,Y 293.026,Z 499.739,A -85,B 0,C 180,E1 -16666.49,E2 -16666.49} C_VEL
LIN {X 0,Y 294.131,Z 489.761,A -85,B 0,C 180,E1 -16667.917,E2 -16667.917} C_VEL
LIN {X 0,Y 295.205,Z 479.495,A -85,B 0,C 180,E1 -16669.108,E2 -16669.108} C_VEL
LIN {X 0,Y 296.405,Z 467.475,A -85,B 0,C 180,E1 -16670.2,E2 -16670.2} C_VEL
LIN {X 0,Y 297.55,Z 453.804,A -85,B 0,C 180,E1 -16671.112,E2 -16671.112} C_VEL
LIN {X 0,Y 298.31,Z 441.055,A -85,B 0,C 180,E1 -16671.69,E2 -16671.69} C_VEL
LIN {X 0,Y 300.103,Z 378.168,A -85,B 0,C 180,E1 -16673.54,E2 -16673.54} C_VEL
LIN {X 0,Y 294.914,Z 333.524,A -85,B 0,C 180,E1 -16675.272,E2 -16675.272} C_VEL
LIN {X 0,Y 295.762,Z 326.218,A -85,B 0,C 180,E1 -16677.221,E2 -16677.221} C_VEL
LIN {X 0,Y 293.867,Z 316.115,A -85,B 0,C 180,E1 -16680.147,E2 -16680.147} C_VEL
LIN {X 0,Y 291.392,Z 304.188,A -85,B 0,C 180,E1 -16683.791,E2 -16683.791} C_VEL
LIN {X 0,Y 291.35,Z 304.191,A -85,B 0,C 180,E1 -16687.246,E2 -16687.246} C_VEL
LIN {X 0,Y 291.288,Z 304.198,A -85,B 0,C 180,E1 -16691.586,E2 -16691.586} C_VEL
LIN {X 0,Y 291.274,Z 304.199,A -85,B 0,C 180,E1 -16695.594,E2 -16695.594} C_VEL
LIN {X 0,Y 291.286,Z 304.2,A -85,B 0,C 180,E1 -16699.349,E2 -16699.349} C_VEL
LIN {X 0,Y 291.371,Z 304.192,A -85,B 0,C 180,E1 -16702.913,E2 -16702.913} C_VEL
LIN {X 0,Y 291.33,Z 304.193,A -85,B 0,C 180,E1 -16706.299,E2 -16706.299} C_VEL
LIN {X 0,Y 291.356,Z 304.19,A -85,B 0,C 180,E1 -16710.265,E2 -16710.265} C_VEL
LIN {X 0,Y 291.345,Z 304.191,A -85,B 0,C 180,E1 -16714.264,E2 -16714.264} C_VEL
LIN {X 0,Y 291.347,Z 304.194,A -85,B 0,C 180,E1 -16717.296,E2 -16717.296} C_VEL
LIN {X 0,Y 291.373,Z 304.187,A -85,B 0,C 180,E1 -16720.263,E2 -16720.263} C_VEL
LIN {X 0,Y 291.481,Z 304.174,A -85,B 0,C 180,E1 -16724.664,E2 -16724.664} C_VEL
LIN {X 0,Y 291.508,Z 304.172,A -85,B 0,C 180,E1 -16728.879,E2 -16728.879} C_VEL
LIN {X 0,Y 291.659,Z 304.154,A -85,B 0,C 180,E1 -16731.686,E2 -16731.686} C_VEL
LIN {X 0,Y 291.599,Z 304.158,A -85,B 0,C 180,E1 -16734.467,E2 -16734.467} C_VEL
LIN {X 0,Y 291.864,Z 304.126,A -85,B 0,C 180,E1 -16738.62,E2 -16738.62} C_VEL
LIN {X 0,Y 291.864,Z 304.13,A -85,B 0,C 180,E1 -16741.379,E2 -16741.379} C_VEL
LIN {X 0,Y 291.7,Z 304.147,A -85,B 0,C 180,E1 -16746.918,E2 -16746.918} C_VEL
LIN {X 0,Y 291.553,Z 304.168,A -85,B 0,C 180,E1 -16749.714,E2 -16749.714} C_VEL
LIN {X 0,Y 291.494,Z 304.175,A -85,B 0,C 180,E1 -16753.951,E2 -16753.951} C_VEL
LIN {X 0,Y 291.403,Z 304.183,A -85,B 0,C 180,E1 -16756.822,E2 -16756.822} C_VEL
LIN {X 0,Y 291.374,Z 304.191,A -85,B 0,C 180,E1 -16759.842,E2 -16759.842} C_VEL
LIN {X 0,Y 291.365,Z 304.19,A -85,B 0,C 180,E1 -16764.208,E2 -16764.208} C_VEL
LIN {X 0,Y 291.405,Z 304.184,A -85,B 0,C 180,E1 -16767.272,E2 -16767.272} C_VEL
LIN {X 0,Y 291.321,Z 304.195,A -85,B 0,C 180,E1 -16770.438,E2 -16770.438} C_VEL
LIN {X 0,Y 291.329,Z 304.196,A -85,B 0,C 180,E1 -16773.699,E2 -16773.699} C_VEL
LIN {X 0,Y 291.367,Z 304.188,A -85,B 0,C 180,E1 -16777.256,E2 -16777.256} C_VEL
LIN {X 0,Y 291.326,Z 304.194,A -85,B 0,C 180,E1 -16780.643,E2 -16780.643} C_VEL
LIN {X 0,Y 291.305,Z 304.197,A -85,B 0,C 180,E1 -16784.398,E2 -16784.398} C_VEL
LIN {X 0,Y 291.371,Z 304.19,A -85,B 0,C 180,E1 -16788.393,E2 -16788.393} C_VEL
LIN {X 0,Y 291.376,Z 304.186,A -85,B 0,C 180,E1 -16791.164,E2 -16791.164} C_VEL
LIN {X 0,Y 291.379,Z 304.188,A -85,B 0,C 180,E1 -16794.63,E2 -16794.63} C_VEL
LIN {X 0,Y 291.364,Z 304.191,A -85,B 0,C 180,E1 -16797.951,E2 -16797.951} C_VEL
LIN {X 0,Y 291.372,Z 304.186,A -85,B 0,C 180,E1 -16801.158,E2 -16801.158} C_VEL
LIN {X 0,Y 291.411,Z 304.188,A -85,B 0,C 180,E1 -16804.272,E2 -16804.272} C_VEL
LIN {X 0,Y 291.385,Z 304.185,A -85,B 0,C 180,E1 -16807.3,E2 -16807.3} C_VEL
LIN {X 0,Y 291.456,Z 304.18,A -85,B 0,C 180,E1 -16810.27,E2 -16810.27} C_VEL
LIN {X 0,Y 291.553,Z 304.168,A -85,B 0,C 180,E1 -16814.623,E2 -16814.623} C_VEL
LIN {X 0,Y 291.535,Z 304.169,A -85,B 0,C 180,E1 -16818.879,E2 -16818.879} C_VEL
LIN {X 0,Y 291.707,Z 304.146,A -85,B 0,C 180,E1 -16821.687,E2 -16821.687} C_VEL
LIN {X 0,Y 291.628,Z 304.16,A -85,B 0,C 180,E1 -16824.467,E2 -16824.467} C_VEL
LIN {X 0,Y 291.887,Z 304.128,A -85,B 0,C 180,E1 -16828.618,E2 -16828.618} C_VEL
LIN {X 0,Y 291.887,Z 304.124,A -85,B 0,C 180,E1 -16831.377,E2 -16831.377} C_VEL
LIN {X 0,Y 291.741,Z 304.145,A -85,B 0,C 180,E1 -16836.915,E2 -16836.915} C_VEL
LIN {X 0,Y 291.624,Z 304.156,A -85,B 0,C 180,E1 -16839.709,E2 -16839.709} C_VEL
LIN {X 0,Y 291.516,Z 304.17,A -85,B 0,C 180,E1 -16843.947,E2 -16843.947} C_VEL
LIN {X 0,Y 291.48,Z 304.178,A -85,B 0,C 180,E1 -16846.814,E2 -16846.814} C_VEL
LIN {X 0,Y 291.474,Z 304.175,A -85,B 0,C 180,E1 -16849.889,E2 -16849.889} C_VEL
LIN {X 0,Y 291.389,Z 304.186,A -85,B 0,C 180,E1 -16854.201,E2 -16854.201} C_VEL
LIN {X 0,Y 291.411,Z 304.186,A -85,B 0,C 180,E1 -16857.267,E2 -16857.267} C_VEL
LIN {X 0,Y 291.321,Z 304.195,A -85,B 0,C 180,E1 -16860.433,E2 -16860.433} C_VEL
LIN {X 0,Y 291.326,Z 304.195,A -85,B 0,C 180,E1 -16863.694,E2 -16863.694} C_VEL
LIN {X 0,Y 291.404,Z 304.186,A -85,B 0,C 180,E1 -16866.696,E2 -16866.696} C_VEL
LIN {X 0,Y 298.818,Z 325.027,A -85,B 0,C 180,E1 -16867.861,E2 -16867.861} C_VEL
LIN {X 0,Y 301.039,Z 331.825,A -85,B 0,C 180,E1 -16868.208,E2 -16868.208} C_VEL
LIN {X 0,Y 298.486,Z 409.941,A -85,B 0,C 180,E1 -16870.498,E2 -16870.498} C_VEL
LIN {X 0,Y 297.999,Z 422.768,A -85,B 0,C 180,E1 -16871.132,E2 -16871.132} C_VEL
LIN {X 0,Y 297.193,Z 435.003,A -85,B 0,C 180,E1 -16871.976,E2 -16871.976} C_VEL
LIN {X 0,Y 296.189,Z 446.807,A -85,B 0,C 180,E1 -16873.06,E2 -16873.06} C_VEL
LIN {X 0,Y 295.075,Z 458.21,A -85,B 0,C 180,E1 -16874.396,E2 -16874.396} C_VEL
LIN {X 0,Y 294.084,Z 467.839,A -85,B 0,C 180,E1 -16875.793,E2 -16875.793} C_VEL
LIN {X 0,Y 292.972,Z 477.815,A -85,B 0,C 180,E1 -16877.572,E2 -16877.572} C_VEL
LIN {X 0,Y 292.001,Z 486.402,A -85,B 0,C 180,E1 -16879.471,E2 -16879.471} C_VEL
LIN {X 0,Y 291.164,Z 494.086,A -85,B 0,C 180,E1 -16881.572,E2 -16881.572} C_VEL
LIN {X 0,Y 290.503,Z 500.245,A -85,B 0,C 180,E1 -16883.693,E2 -16883.693} C_VEL
LIN {X 0,Y 290.053,Z 505.652,A -85,B 0,C 180,E1 -16886.132,E2 -16886.132} C_VEL
LIN {X 0,Y 289.704,Z 508.905,A -85,B 0,C 180,E1 -16888.097,E2 -16888.097} C_VEL
LIN {X 0,Y 289.523,Z 510.498,A -85,B 0,C 180,E1 -16889.353,E2 -16889.353} C_VEL
LIN {X 0,Y 289.492,Z 512.033,A -85,B 0,C 180,E1 -16890.953,E2 -16890.953} C_VEL
LIN {X 0,Y 289.477,Z 512.955,A -85,B 0,C 180,E1 -16892.531,E2 -16892.531} C_VEL
LIN {X 0,Y 289.6,Z 513.39,A -85,B 0,C 180,E1 -16894.099,E2 -16894.099} C_VEL
LIN {X 0,Y 289.838,Z 513.254,A -85,B 0,C 180,E1 -16895.657,E2 -16895.657} C_VEL
LIN {X 0,Y 290.152,Z 512.633,A -85,B 0,C 180,E1 -16897.199,E2 -16897.199} C_VEL
LIN {X 0,Y 290.609,Z 511.505,A -85,B 0,C 180,E1 -16898.731,E2 -16898.731} C_VEL
LIN {X 0,Y 291.459,Z 508.831,A -85,B 0,C 180,E1 -16901.012,E2 -16901.012} C_VEL
LIN {X 0,Y 292.539,Z 505.008,A -85,B 0,C 180,E1 -16903.245,E2 -16903.245} C_VEL
LIN {X 0,Y 293.969,Z 499.901,A -85,B 0,C 180,E1 -16905.462,E2 -16905.462} C_VEL
LIN {X 0,Y 295.739,Z 493.355,A -85,B 0,C 180,E1 -16907.651,E2 -16907.651} C_VEL
LIN {X 0,Y 296.331,Z 491.002,A -85,B 0,C 180,E1 -16908.313,E2 -16908.313} C_VEL
LIN {X 0,Y 296.557,Z 487.689,A -85,B 0,C 180,E1 -16909.259,E2 -16909.259} C_VEL
LIN {X 0,Y 295.361,Z 482.123,A -85,B 0,C 180,E1 -16910.833,E2 -16910.833} C_VEL
LIN {X 0,Y 294.291,Z 476.062,A -85,B 0,C 180,E1 -16912.332,E2 -16912.332} C_VEL
LIN {X 0,Y 294.688,Z 471.884,A -85,B 0,C 180,E1 -16913.144,E2 -16913.144} C_VEL
LIN {X 0,Y 296.914,Z 461.16,A -85,B 0,C 180,E1 -16914.756,E2 -16914.756} C_VEL
LIN {X 0,Y 298.98,Z 449.675,A -85,B 0,C 180,E1 -16916.126,E2 -16916.126} C_VEL
LIN {X 0,Y 300.773,Z 437.535,A -85,B 0,C 180,E1 -16917.238,E2 -16917.238} C_VEL
LIN {X 0,Y 302.311,Z 423.496,A -85,B 0,C 180,E1 -16918.201,E2 -16918.201} C_VEL
LIN {X 0,Y 303.345,Z 410.315,A -85,B 0,C 180,E1 -16918.8,E2 -16918.8} C_VEL
LIN {X 0,Y 307.334,Z 344.801,A -85,B 0,C 180,E1 -16920.859,E2 -16920.859} C_VEL
LIN {X 0,Y 302.145,Z 333.419,A -85,B 0,C 180,E1 -16922.217,E2 -16922.217} C_VEL
LIN {X 0,Y 297.375,Z 324.758,A -85,B 0,C 180,E1 -16923.494,E2 -16923.494} C_VEL
LIN {X 0,Y 292.686,Z 317.845,A -85,B 0,C 180,E1 -16924.778,E2 -16924.778} C_VEL
LIN {X 0,Y 286.443,Z 308.897,A -85,B 0,C 180,E1 -16926.658,E2 -16926.658} C_VEL
LIN {X 0,Y 285.061,Z 306.719,A -85,B 0,C 180,E1 -16927.171,E2 -16927.171} C_VEL
LIN {X 0,Y 284.601,Z 305.032,A -85,B 0,C 180,E1 -16927.985,E2 -16927.985} C_VEL
LIN {X 0,Y 284.432,Z 305.051,A -85,B 0,C 180,E1 -16932.85,E2 -16932.85} C_VEL
LIN {X 0,Y 284.372,Z 305.059,A -85,B 0,C 180,E1 -16935.775,E2 -16935.775} C_VEL
LIN {X 0,Y 284.288,Z 305.065,A -85,B 0,C 180,E1 -16940.25,E2 -16940.25} C_VEL
LIN {X 0,Y 284.297,Z 305.068,A -85,B 0,C 180,E1 -16943.861,E2 -16943.861} C_VEL
LIN {X 0,Y 284.346,Z 305.066,A -85,B 0,C 180,E1 -16947.17,E2 -16947.17} C_VEL
LIN {X 0,Y 284.255,Z 305.071,A -85,B 0,C 180,E1 -16951.28,E2 -16951.28} C_VEL
LIN {X 0,Y 284.314,Z 305.066,A -85,B 0,C 180,E1 -16955.352,E2 -16955.352} C_VEL
LIN {X 0,Y 284.299,Z 305.071,A -85,B 0,C 180,E1 -16958.172,E2 -16958.172} C_VEL
LIN {X 0,Y 284.247,Z 305.073,A -85,B 0,C 180,E1 -16962.129,E2 -16962.129} C_VEL
LIN {X 0,Y 284.235,Z 305.078,A -85,B 0,C 180,E1 -16966.194,E2 -16966.194} C_VEL
LIN {X 0,Y 284.275,Z 305.22,A -85,B 0,C 180,E1 -16967.347,E2 -16967.347} C_VEL
LIN {X 0,Y 286.47,Z 311.396,A -85,B 0,C 180,E1 -16970.375,E2 -16970.375} C_VEL
LIN {X 0,Y 289.181,Z 319.818,A -85,B 0,C 180,E1 -16973.958,E2 -16973.958} C_VEL
LIN {X 0,Y 290.972,Z 326.265,A -85,B 0,C 180,E1 -16976.337,E2 -16976.337} C_VEL
LIN {X 0,Y 294.736,Z 333.701,A -85,B 0,C 180,E1 -16977.475,E2 -16977.475} C_VEL
LIN {X 0,Y 298.568,Z 341.516,A -85,B 0,C 180,E1 -16978.557,E2 -16978.557} C_VEL
LIN {X 0,Y 300.536,Z 346.552,A -85,B 0,C 180,E1 -16979.136,E2 -16979.136} C_VEL
LIN {X 0,Y 303.432,Z 363.559,A -85,B 0,C 180,E1 -16980.359,E2 -16980.359} C_VEL
LIN {X 0,Y 305.416,Z 381.215,A -85,B 0,C 180,E1 -16981.397,E2 -16981.397} C_VEL
LIN {X 0,Y 305.134,Z 389.612,A -85,B 0,C 180,E1 -16981.694,E2 -16981.694} C_VEL
LIN {X 0,Y 302.149,Z 439.402,A -85,B 0,C 180,E1 -16983.266,E2 -16983.266} C_VEL
LIN {X 0,Y 300.687,Z 453.008,A -85,B 0,C 180,E1 -16983.92,E2 -16983.92} C_VEL
LIN {X 0,Y 298.813,Z 465.582,A -85,B 0,C 180,E1 -16984.772,E2 -16984.772} C_VEL
LIN {X 0,Y 296.606,Z 477.731,A -85,B 0,C 180,E1 -16985.88,E2 -16985.88} C_VEL
LIN {X 0,Y 294.409,Z 488.801,A -85,B 0,C 180,E1 -16987.18,E2 -16987.18} C_VEL
LIN {X 0,Y 292.177,Z 498.956,A -85,B 0,C 180,E1 -16988.67,E2 -16988.67} C_VEL
LIN {X 0,Y 289.727,Z 509.065,A -85,B 0,C 180,E1 -16990.521,E2 -16990.521} C_VEL
LIN {X 0,Y 287.579,Z 518.064,A -85,B 0,C 180,E1 -16992.574,E2 -16992.574} C_VEL
LIN {X 0,Y 285.919,Z 525.39,A -85,B 0,C 180,E1 -16994.682,E2 -16994.682} C_VEL
LIN {X 0,Y 284.144,Z 532.134,A -85,B 0,C 180,E1 -16997.142,E2 -16997.142} C_VEL
LIN {X 0,Y 283.297,Z 536.631,A -85,B 0,C 180,E1 -16999.281,E2 -16999.281} C_VEL
LIN {X 0,Y 282.757,Z 540.067,A -85,B 0,C 180,E1 -17001.427,E2 -17001.427} C_VEL
LIN {X 0,Y 282.505,Z 541.817,A -85,B 0,C 180,E1 -17002.858,E2 -17002.858} C_VEL
LIN {X 0,Y 282.438,Z 543.246,A -85,B 0,C 180,E1 -17004.468,E2 -17004.468} C_VEL
LIN {X 0,Y 282.477,Z 544.454,A -85,B 0,C 180,E1 -17007.15,E2 -17007.15} C_VEL
LIN {X 0,Y 282.535,Z 544.509,A -85,B 0,C 180,E1 -17008.577,E2 -17008.577} C_VEL
LIN {X 0,Y 282.752,Z 544.128,A -85,B 0,C 180,E1 -17010.002,E2 -17010.002} C_VEL
LIN {X 0,Y 282.626,Z 543.272,A -85,B 0,C 180,E1 -17011.427,E2 -17011.427} C_VEL
LIN {X 0,Y 282.543,Z 541.992,A -85,B 0,C 180,E1 -17012.854,E2 -17012.854} C_VEL
LIN {X 0,Y 282.598,Z 539.204,A -85,B 0,C 180,E1 -17014.995,E2 -17014.995} C_VEL
LIN {X 0,Y 282.674,Z 535.288,A -85,B 0,C 180,E1 -17017.143,E2 -17017.143} C_VEL
LIN {X 0,Y 282.87,Z 530.143,A -85,B 0,C 180,E1 -17019.295,E2 -17019.295} C_VEL
LIN {X 0,Y 283.345,Z 523.608,A -85,B 0,C 180,E1 -17021.446,E2 -17021.446} C_VEL
LIN {X 0,Y 284.259,Z 515.397,A -85,B 0,C 180,E1 -17023.585,E2 -17023.585} C_VEL
LIN {X 0,Y 285.247,Z 507.004,A -85,B 0,C 180,E1 -17025.359,E2 -17025.359} C_VEL
LIN {X 0,Y 286.1,Z 498.666,A -85,B 0,C 180,E1 -17026.819,E2 -17026.819} C_VEL
LIN {X 0,Y 287.362,Z 487.971,A -85,B 0,C 180,E1 -17028.354,E2 -17028.354} C_VEL
LIN {X 0,Y 288.728,Z 475.598,A -85,B 0,C 180,E1 -17029.739,E2 -17029.739} C_VEL
LIN {X 0,Y 289.88,Z 463.675,A -85,B 0,C 180,E1 -17030.768,E2 -17030.768} C_VEL
LIN {X 0,Y 290.815,Z 450.841,A -85,B 0,C 180,E1 -17031.579,E2 -17031.579} C_VEL
LIN {X 0,Y 291.501,Z 437.768,A -85,B 0,C 180,E1 -17032.13,E2 -17032.13} C_VEL
LIN {X 0,Y 293.313,Z 379.24,A -85,B 0,C 180,E1 -17033.885,E2 -17033.885} C_VEL
LIN {X 0,Y 288.067,Z 333.113,A -85,B 0,C 180,E1 -17035.742,E2 -17035.742} C_VEL
LIN {X 0,Y 288.735,Z 327.931,A -85,B 0,C 180,E1 -17037.154,E2 -17037.154} C_VEL
LIN {X 0,Y 287.58,Z 320.726,A -85,B 0,C 180,E1 -17039.259,E2 -17039.259} C_VEL
LIN {X 0,Y 284.863,Z 307.536,A -85,B 0,C 180,E1 -17043.292,E2 -17043.292} C_VEL
LIN {X 0,Y 284.338,Z 305.067,A -85,B 0,C 180,E1 -17044.107,E2 -17044.107} C_VEL
LIN {X 0,Y 284.261,Z 305.074,A -85,B 0,C 180,E1 -17048.175,E2 -17048.175} C_VEL
LIN {X 0,Y 284.23,Z 305.078,A -85,B 0,C 180,E1 -17052.115,E2 -17052.115} C_VEL
LIN {X 0,Y 284.229,Z 305.077,A -85,B 0,C 180,E1 -17056.183,E2 -17056.183} C_VEL
LIN {X 0,Y 284.276,Z 305.072,A -85,B 0,C 180,E1 -17060.028,E2 -17060.028} C_VEL
LIN {X 0,Y 284.305,Z 305.068,A -85,B 0,C 180,E1 -17063.609,E2 -17063.609} C_VEL
LIN {X 0,Y 284.275,Z 305.075,A -85,B 0,C 180,E1 -17067.195,E2 -17067.195} C_VEL
LIN {X 0,Y 284.328,Z 305.065,A -85,B 0,C 180,E1 -17070.372,E2 -17070.372} C_VEL
LIN {X 0,Y 284.294,Z 305.071,A -85,B 0,C 180,E1 -17073.577,E2 -17073.577} C_VEL
LIN {X 0,Y 284.312,Z 305.068,A -85,B 0,C 180,E1 -17076.702,E2 -17076.702} C_VEL
LIN {X 0,Y 284.314,Z 305.072,A -85,B 0,C 180,E1 -17081.255,E2 -17081.255} C_VEL
LIN {X 0,Y 284.444,Z 305.051,A -85,B 0,C 180,E1 -17085.695,E2 -17085.695} C_VEL
LIN {X 0,Y 284.496,Z 305.044,A -85,B 0,C 180,E1 -17090.041,E2 -17090.041} C_VEL
LIN {X 0,Y 284.66,Z 305.025,A -85,B 0,C 180,E1 -17092.908,E2 -17092.908} C_VEL
LIN {X 0,Y 284.831,Z 305.002,A -85,B 0,C 180,E1 -17098.585,E2 -17098.585} C_VEL
LIN {X 0,Y 284.831,Z 305.007,A -85,B 0,C 180,E1 -17101.413,E2 -17101.413} C_VEL
LIN {X 0,Y 284.653,Z 305.026,A -85,B 0,C 180,E1 -17107.09,E2 -17107.09} C_VEL
LIN {X 0,Y 284.498,Z 305.045,A -85,B 0,C 180,E1 -17109.957,E2 -17109.957} C_VEL
LIN {X 0,Y 284.443,Z 305.051,A -85,B 0,C 180,E1 -17114.304,E2 -17114.304} C_VEL
LIN {X 0,Y 284.308,Z 305.066,A -85,B 0,C 180,E1 -17118.744,E2 -17118.744} C_VEL
LIN {X 0,Y 284.315,Z 305.068,A -85,B 0,C 180,E1 -17123.297,E2 -17123.297} C_VEL
LIN {X 0,Y 284.38,Z 305.058,A -85,B 0,C 180,E1 -17127.173,E2 -17127.173} C_VEL
LIN {X 0,Y 284.28,Z 305.072,A -85,B 0,C 180,E1 -17131.275,E2 -17131.275} C_VEL
LIN {X 0,Y 284.328,Z 305.065,A -85,B 0,C 180,E1 -17135.348,E2 -17135.348} C_VEL
LIN {X 0,Y 284.306,Z 305.071,A -85,B 0,C 180,E1 -17138.169,E2 -17138.169} C_VEL
LIN {X 0,Y 284.262,Z 305.077,A -85,B 0,C 180,E1 -17142.126,E2 -17142.126} C_VEL
LIN {X 0,Y 284.298,Z 305.073,A -85,B 0,C 180,E1 -17146.2,E2 -17146.2} C_VEL
LIN {X 0,Y 284.344,Z 305.067,A -85,B 0,C 180,E1 -17150.014,E2 -17150.014} C_VEL
LIN {X 0,Y 284.348,Z 305.062,A -85,B 0,C 180,E1 -17153.618,E2 -17153.618} C_VEL
LIN {X 0,Y 284.301,Z 305.068,A -85,B 0,C 180,E1 -17157.19,E2 -17157.19} C_VEL
LIN {X 0,Y 284.35,Z 305.065,A -85,B 0,C 180,E1 -17160.376,E2 -17160.376} C_VEL
LIN {X 0,Y 284.372,Z 305.06,A -85,B 0,C 180,E1 -17163.586,E2 -17163.586} C_VEL
LIN {X 0,Y 284.365,Z 305.062,A -85,B 0,C 180,E1 -17166.707,E2 -17166.707} C_VEL
LIN {X 0,Y 284.401,Z 305.055,A -85,B 0,C 180,E1 -17171.261,E2 -17171.261} C_VEL
LIN {X 0,Y 284.49,Z 305.05,A -85,B 0,C 180,E1 -17174.458,E2 -17174.458} C_VEL
LIN {X 0,Y 284.486,Z 305.049,A -85,B 0,C 180,E1 -17178.6,E2 -17178.6} C_VEL
LIN {X 0,Y 284.657,Z 305.024,A -85,B 0,C 180,E1 -17181.48,E2 -17181.48} C_VEL
LIN {X 0,Y 284.599,Z 305.034,A -85,B 0,C 180,E1 -17184.33,E2 -17184.33} C_VEL
LIN {X 0,Y 284.853,Z 305.004,A -85,B 0,C 180,E1 -17188.584,E2 -17188.584} C_VEL
LIN {X 0,Y 284.853,Z 305,A -85,B 0,C 180,E1 -17191.411,E2 -17191.411} C_VEL
LIN {X 0,Y 284.693,Z 305.022,A -85,B 0,C 180,E1 -17197.087,E2 -17197.087} C_VEL
LIN {X 0,Y 284.561,Z 305.036,A -85,B 0,C 180,E1 -17199.952,E2 -17199.952} C_VEL
LIN {X 0,Y 284.475,Z 305.048,A -85,B 0,C 180,E1 -17204.299,E2 -17204.299} C_VEL
LIN {X 0,Y 284.421,Z 305.055,A -85,B 0,C 180,E1 -17207.244,E2 -17207.244} C_VEL
LIN {X 0,Y 284.409,Z 305.056,A -85,B 0,C 180,E1 -17210.235,E2 -17210.235} C_VEL
LIN {X 0,Y 284.358,Z 305.061,A -85,B 0,C 180,E1 -17213.872,E2 -17213.872} C_VEL
LIN {X 0,Y 284.385,Z 305.062,A -85,B 0,C 180,E1 -17217.17,E2 -17217.17} C_VEL
LIN {X 0,Y 284.278,Z 305.075,A -85,B 0,C 180,E1 -17221.27,E2 -17221.27} C_VEL
LIN {X 0,Y 284.326,Z 305.067,A -85,B 0,C 180,E1 -17225.798,E2 -17225.798} C_VEL
LIN {X 0,Y 284.336,Z 305.07,A -85,B 0,C 180,E1 -17226.269,E2 -17226.269} C_VEL
LIN {X 0,Y 291.997,Z 326.35,A -85,B 0,C 180,E1 -17227.473,E2 -17227.473} C_VEL
LIN {X 0,Y 294.338,Z 333.756,A -85,B 0,C 180,E1 -17227.857,E2 -17227.857} C_VEL
LIN {X 0,Y 291.628,Z 410.242,A -85,B 0,C 180,E1 -17230.154,E2 -17230.154} C_VEL
LIN {X 0,Y 291.096,Z 423.474,A -85,B 0,C 180,E1 -17230.826,E2 -17230.826} C_VEL
LIN {X 0,Y 290.244,Z 435.868,A -85,B 0,C 180,E1 -17231.71,E2 -17231.71} C_VEL
LIN {X 0,Y 289.205,Z 447.996,A -85,B 0,C 180,E1 -17232.869,E2 -17232.869} C_VEL
LIN {X 0,Y 288.044,Z 459.103,A -85,B 0,C 180,E1 -17234.217,E2 -17234.217} C_VEL
LIN {X 0,Y 286.984,Z 469.207,A -85,B 0,C 180,E1 -17235.739,E2 -17235.739} C_VEL
LIN {X 0,Y 285.889,Z 478.705,A -85,B 0,C 180,E1 -17237.508,E2 -17237.508} C_VEL
LIN {X 0,Y 284.817,Z 487.822,A -85,B 0,C 180,E1 -17239.608,E2 -17239.608} C_VEL
LIN {X 0,Y 283.964,Z 495.336,A -85,B 0,C 180,E1 -17241.777,E2 -17241.777} C_VEL
LIN {X 0,Y 283.242,Z 502.095,A -85,B 0,C 180,E1 -17244.287,E2 -17244.287} C_VEL
LIN {X 0,Y 282.834,Z 507.279,A -85,B 0,C 180,E1 -17246.862,E2 -17246.862} C_VEL
LIN {X 0,Y 282.558,Z 509.745,A -85,B 0,C 180,E1 -17248.512,E2 -17248.512} C_VEL
LIN {X 0,Y 282.394,Z 511.979,A -85,B 0,C 180,E1 -17250.566,E2 -17250.566} C_VEL
LIN {X 0,Y 282.433,Z 513.636,A -85,B 0,C 180,E1 -17253.391,E2 -17253.391} C_VEL
LIN {X 0,Y 282.625,Z 513.812,A -85,B 0,C 180,E1 -17254.993,E2 -17254.993} C_VEL
LIN {X 0,Y 282.968,Z 513.448,A -85,B 0,C 180,E1 -17256.755,E2 -17256.755} C_VEL
LIN {X 0,Y 283.332,Z 512.664,A -85,B 0,C 180,E1 -17258.157,E2 -17258.157} C_VEL
LIN {X 0,Y 284.015,Z 510.973,A -85,B 0,C 180,E1 -17260.082,E2 -17260.082} C_VEL
LIN {X 0,Y 284.836,Z 508.411,A -85,B 0,C 180,E1 -17262.037,E2 -17262.037} C_VEL
LIN {X 0,Y 286.142,Z 504.269,A -85,B 0,C 180,E1 -17264.326,E2 -17264.326} C_VEL
LIN {X 0,Y 287.782,Z 498.759,A -85,B 0,C 180,E1 -17266.586,E2 -17266.586} C_VEL
LIN {X 0,Y 289.736,Z 491.754,A -85,B 0,C 180,E1 -17268.811,E2 -17268.811} C_VEL
LIN {X 0,Y 291.833,Z 483.737,A -85,B 0,C 180,E1 -17270.835,E2 -17270.835} C_VEL
LIN {X 0,Y 294.015,Z 474.85,A -85,B 0,C 180,E1 -17272.619,E2 -17272.619} C_VEL
LIN {X 0,Y 294.688,Z 471.884,A -85,B 0,C 180,E1 -17273.144,E2 -17273.144} C_VEL
LIN {X 0,Y 295.106,Z 467.579,A -85,B 0,C 180,E1 -17273.928,E2 -17273.928} C_VEL
LIN {X 0,Y 294.162,Z 460.502,A -85,B 0,C 180,E1 -17275.271,E2 -17275.271} C_VEL
LIN {X 0,Y 293.163,Z 452.981,A -85,B 0,C 180,E1 -17276.509,E2 -17276.509} C_VEL
LIN {X 0,Y 293.46,Z 447.989,A -85,B 0,C 180,E1 -17277.116,E2 -17277.116} C_VEL
LIN {X 0,Y 295.282,Z 435.999,A -85,B 0,C 180,E1 -17278.193,E2 -17278.193} C_VEL
LIN {X 0,Y 296.736,Z 422.979,A -85,B 0,C 180,E1 -17279.068,E2 -17279.068} C_VEL
LIN {X 0,Y 297.815,Z 409.659,A -85,B 0,C 180,E1 -17279.663,E2 -17279.663} C_VEL
LIN {X 0,Y 301.786,Z 347.234,A -85,B 0,C 180,E1 -17281.669,E2 -17281.669} C_VEL
LIN {X 0,Y 297.642,Z 337.845,A -85,B 0,C 180,E1 -17282.834,E2 -17282.834} C_VEL
LIN {X 0,Y 293.051,Z 329.418,A -85,B 0,C 180,E1 -17284.126,E2 -17284.126} C_VEL
LIN {X 0,Y 288.25,Z 322.23,A -85,B 0,C 180,E1 -17285.521,E2 -17285.521} C_VEL
LIN {X 0,Y 283.074,Z 314.606,A -85,B 0,C 180,E1 -17287.176,E2 -17287.176} C_VEL
LIN {X 0,Y 279.735,Z 310.194,A -85,B 0,C 180,E1 -17288.307,E2 -17288.307} C_VEL
LIN {X 0,Y 277.979,Z 307.601,A -85,B 0,C 180,E1 -17289.029,E2 -17289.029} C_VEL
LIN {X 0,Y 277.453,Z 305.922,A -85,B 0,C 180,E1 -17289.984,E2 -17289.984} C_VEL
LIN {X 0,Y 277.37,Z 305.93,A -85,B 0,C 180,E1 -17294.678,E2 -17294.678} C_VEL
LIN {X 0,Y 277.247,Z 305.948,A -85,B 0,C 180,E1 -17299.242,E2 -17299.242} C_VEL
LIN {X 0,Y 277.26,Z 305.944,A -85,B 0,C 180,E1 -17303.928,E2 -17303.928} C_VEL
LIN {X 0,Y 277.277,Z 305.947,A -85,B 0,C 180,E1 -17307.502,E2 -17307.502} C_VEL
LIN {X 0,Y 277.219,Z 305.955,A -85,B 0,C 180,E1 -17310.477,E2 -17310.477} C_VEL
LIN {X 0,Y 277.218,Z 305.948,A -85,B 0,C 180,E1 -17313.901,E2 -17313.901} C_VEL
LIN {X 0,Y 277.25,Z 305.944,A -85,B 0,C 180,E1 -17317.473,E2 -17317.473} C_VEL
LIN {X 0,Y 277.187,Z 305.958,A -85,B 0,C 180,E1 -17321.241,E2 -17321.241} C_VEL
LIN {X 0,Y 277.191,Z 306.077,A -85,B 0,C 180,E1 -17325.41,E2 -17325.41} C_VEL
LIN {X 0,Y 278.322,Z 308.918,A -85,B 0,C 180,E1 -17327.079,E2 -17327.079} C_VEL
LIN {X 0,Y 280.561,Z 315.448,A -85,B 0,C 180,E1 -17330.38,E2 -17330.38} C_VEL
LIN {X 0,Y 283.033,Z 323.283,A -85,B 0,C 180,E1 -17333.815,E2 -17333.815} C_VEL
LIN {X 0,Y 283.65,Z 325.399,A -85,B 0,C 180,E1 -17334.622,E2 -17334.622} C_VEL
LIN {X 0,Y 286.587,Z 330.699,A -85,B 0,C 180,E1 -17335.6,E2 -17335.6} C_VEL
LIN {X 0,Y 290.277,Z 337.883,A -85,B 0,C 180,E1 -17336.766,E2 -17336.766} C_VEL
LIN {X 0,Y 294.223,Z 346.373,A -85,B 0,C 180,E1 -17337.968,E2 -17337.968} C_VEL
LIN {X 0,Y 295.561,Z 349.792,A -85,B 0,C 180,E1 -17338.377,E2 -17338.377} C_VEL
LIN {X 0,Y 298.166,Z 366.051,A -85,B 0,C 180,E1 -17339.584,E2 -17339.584} C_VEL
LIN {X 0,Y 299.832,Z 382.065,A -85,B 0,C 180,E1 -17340.558,E2 -17340.558} C_VEL
LIN {X 0,Y 299.814,Z 386.976,A -85,B 0,C 180,E1 -17340.762,E2 -17340.762} C_VEL
LIN {X 0,Y 296.504,Z 438.786,A -85,B 0,C 180,E1 -17342.428,E2 -17342.428} C_VEL
LIN {X 0,Y 294.994,Z 452.271,A -85,B 0,C 180,E1 -17343.091,E2 -17343.091} C_VEL
LIN {X 0,Y 293.143,Z 463.837,A -85,B 0,C 180,E1 -17343.867,E2 -17343.867} C_VEL
LIN {X 0,Y 290.858,Z 476.194,A -85,B 0,C 180,E1 -17344.99,E2 -17344.99} C_VEL
LIN {X 0,Y 288.508,Z 487.459,A -85,B 0,C 180,E1 -17346.306,E2 -17346.306} C_VEL
LIN {X 0,Y 286.077,Z 497.802,A -85,B 0,C 180,E1 -17347.813,E2 -17347.813} C_VEL
LIN {X 0,Y 283.966,Z 506.354,A -85,B 0,C 180,E1 -17349.353,E2 -17349.353} C_VEL
LIN {X 0,Y 281.522,Z 515.618,A -85,B 0,C 180,E1 -17351.415,E2 -17351.415} C_VEL
LIN {X 0,Y 279.642,Z 523.345,A -85,B 0,C 180,E1 -17353.581,E2 -17353.581} C_VEL
LIN {X 0,Y 277.72,Z 530.486,A -85,B 0,C 180,E1 -17356.093,E2 -17356.093} C_VEL
LIN {X 0,Y 276.533,Z 535.252,A -85,B 0,C 180,E1 -17358.273,E2 -17358.273} C_VEL
LIN {X 0,Y 275.859,Z 538.927,A -85,B 0,C 180,E1 -17360.471,E2 -17360.471} C_VEL
LIN {X 0,Y 275.452,Z 541.596,A -85,B 0,C 180,E1 -17362.674,E2 -17362.674} C_VEL
LIN {X 0,Y 275.347,Z 543.078,A -85,B 0,C 180,E1 -17364.534,E2 -17364.534} C_VEL
LIN {X 0,Y 275.401,Z 544.065,A -85,B 0,C 180,E1 -17367.077,E2 -17367.077} C_VEL
LIN {X 0,Y 275.449,Z 544.058,A -85,B 0,C 180,E1 -17368.54,E2 -17368.54} C_VEL
LIN {X 0,Y 275.667,Z 543.6,A -85,B 0,C 180,E1 -17370.002,E2 -17370.002} C_VEL
LIN {X 0,Y 275.539,Z 542.697,A -85,B 0,C 180,E1 -17371.464,E2 -17371.464} C_VEL
LIN {X 0,Y 275.472,Z 541.369,A -85,B 0,C 180,E1 -17372.927,E2 -17372.927} C_VEL
LIN {X 0,Y 275.545,Z 538.173,A -85,B 0,C 180,E1 -17375.322,E2 -17375.322} C_VEL
LIN {X 0,Y 275.6,Z 534.454,A -85,B 0,C 180,E1 -17377.327,E2 -17377.327} C_VEL
LIN {X 0,Y 275.891,Z 528.148,A -85,B 0,C 180,E1 -17379.902,E2 -17379.902} C_VEL
LIN {X 0,Y 276.5,Z 521.213,A -85,B 0,C 180,E1 -17382.106,E2 -17382.106} C_VEL
LIN {X 0,Y 277.299,Z 514.12,A -85,B 0,C 180,E1 -17383.933,E2 -17383.933} C_VEL
LIN {X 0,Y 278.29,Z 505.551,A -85,B 0,C 180,E1 -17385.753,E2 -17385.753} C_VEL
LIN {X 0,Y 279.378,Z 496.347,A -85,B 0,C 180,E1 -17387.351,E2 -17387.351} C_VEL
LIN {X 0,Y 280.778,Z 484.551,A -85,B 0,C 180,E1 -17388.99,E2 -17388.99} C_VEL
LIN {X 0,Y 281.961,Z 473.23,A -85,B 0,C 180,E1 -17390.233,E2 -17390.233} C_VEL
LIN {X 0,Y 283.15,Z 460.593,A -85,B 0,C 180,E1 -17391.285,E2 -17391.285} C_VEL
LIN {X 0,Y 284.203,Z 446.814,A -85,B 0,C 180,E1 -17392.107,E2 -17392.107} C_VEL
LIN {X 0,Y 284.743,Z 432.816,A -85,B 0,C 180,E1 -17392.637,E2 -17392.637} C_VEL
LIN {X 0,Y 286.483,Z 379.661,A -85,B 0,C 180,E1 -17394.273,E2 -17394.273} C_VEL
LIN {X 0,Y 281.223,Z 332.815,A -85,B 0,C 180,E1 -17396.182,E2 -17396.182} C_VEL
LIN {X 0,Y 281.681,Z 328.175,A -85,B 0,C 180,E1 -17397.489,E2 -17397.489} C_VEL
LIN {X 0,Y 280.103,Z 319.502,A -85,B 0,C 180,E1 -17400.119,E2 -17400.119} C_VEL
LIN {X 0,Y 277.655,Z 307.683,A -85,B 0,C 180,E1 -17403.838,E2 -17403.838} C_VEL
LIN {X 0,Y 277.277,Z 305.947,A -85,B 0,C 180,E1 -17404.439,E2 -17404.439} C_VEL
LIN {X 0,Y 277.22,Z 305.951,A -85,B 0,C 180,E1 -17408.195,E2 -17408.195} C_VEL
LIN {X 0,Y 277.186,Z 305.958,A -85,B 0,C 180,E1 -17412.667,E2 -17412.667} C_VEL
LIN {X 0,Y 277.182,Z 305.958,A -85,B 0,C 180,E1 -17416.796,E2 -17416.796} C_VEL
LIN {X 0,Y 277.207,Z 305.955,A -85,B 0,C 180,E1 -17420.666,E2 -17420.666} C_VEL
LIN {X 0,Y 277.265,Z 305.945,A -85,B 0,C 180,E1 -17424.338,E2 -17424.338} C_VEL
LIN {X 0,Y 277.217,Z 305.951,A -85,B 0,C 180,E1 -17427.832,E2 -17427.832} C_VEL
LIN {X 0,Y 277.231,Z 305.953,A -85,B 0,C 180,E1 -17431.205,E2 -17431.205} C_VEL
LIN {X 0,Y 277.234,Z 305.949,A -85,B 0,C 180,E1 -17434.471,E2 -17434.471} C_VEL
LIN {X 0,Y 277.243,Z 305.948,A -85,B 0,C 180,E1 -17437.65,E2 -17437.65} C_VEL
LIN {X 0,Y 277.268,Z 305.946,A -85,B 0,C 180,E1 -17440.76,E2 -17440.76} C_VEL
LIN {X 0,Y 277.391,Z 305.933,A -85,B 0,C 180,E1 -17445.323,E2 -17445.323} C_VEL
LIN {X 0,Y 277.437,Z 305.925,A -85,B 0,C 180,E1 -17449.785,E2 -17449.785} C_VEL
LIN {X 0,Y 277.615,Z 305.901,A -85,B 0,C 180,E1 -17452.727,E2 -17452.727} C_VEL
LIN {X 0,Y 277.797,Z 305.879,A -85,B 0,C 180,E1 -17458.55,E2 -17458.55} C_VEL
LIN {X 0,Y 277.797,Z 305.883,A -85,B 0,C 180,E1 -17461.449,E2 -17461.449} C_VEL
LIN {X 0,Y 277.609,Z 305.905,A -85,B 0,C 180,E1 -17467.271,E2 -17467.271} C_VEL
LIN {X 0,Y 277.441,Z 305.922,A -85,B 0,C 180,E1 -17470.213,E2 -17470.213} C_VEL
LIN {X 0,Y 277.39,Z 305.929,A -85,B 0,C 180,E1 -17474.676,E2 -17474.676} C_VEL
LIN {X 0,Y 277.264,Z 305.945,A -85,B 0,C 180,E1 -17479.239,E2 -17479.239} C_VEL
LIN {X 0,Y 277.28,Z 305.947,A -85,B 0,C 180,E1 -17483.924,E2 -17483.924} C_VEL
LIN {X 0,Y 277.309,Z 305.941,A -85,B 0,C 180,E1 -17487.505,E2 -17487.505} C_VEL
LIN {X 0,Y 277.259,Z 305.946,A -85,B 0,C 180,E1 -17490.482,E2 -17490.482} C_VEL
LIN {X 0,Y 277.233,Z 305.953,A -85,B 0,C 180,E1 -17493.897,E2 -17493.897} C_VEL
LIN {X 0,Y 277.259,Z 305.946,A -85,B 0,C 180,E1 -17497.47,E2 -17497.47} C_VEL
LIN {X 0,Y 277.202,Z 305.953,A -85,B 0,C 180,E1 -17501.237,E2 -17501.237} C_VEL
LIN {X 0,Y 277.221,Z 305.949,A -85,B 0,C 180,E1 -17505.221,E2 -17505.221} C_VEL
LIN {X 0,Y 277.285,Z 305.943,A -85,B 0,C 180,E1 -17509.496,E2 -17509.496} C_VEL
LIN {X 0,Y 277.282,Z 305.943,A -85,B 0,C 180,E1 -17512.535,E2 -17512.535} C_VEL
LIN {X 0,Y 277.248,Z 305.951,A -85,B 0,C 180,E1 -17516.106,E2 -17516.106} C_VEL
LIN {X 0,Y 277.257,Z 305.946,A -85,B 0,C 180,E1 -17519.539,E2 -17519.539} C_VEL
LIN {X 0,Y 277.352,Z 305.934,A -85,B 0,C 180,E1 -17522.864,E2 -17522.864} C_VEL
LIN {X 0,Y 277.325,Z 305.94,A -85,B 0,C 180,E1 -17526.079,E2 -17526.079} C_VEL
LIN {X 0,Y 277.343,Z 305.937,A -85,B 0,C 180,E1 -17530.766,E2 -17530.766} C_VEL
LIN {X 0,Y 277.433,Z 305.924,A -85,B 0,C 180,E1 -17535.325,E2 -17535.325} C_VEL
LIN {X 0,Y 277.505,Z 305.915,A -85,B 0,C 180,E1 -17539.787,E2 -17539.787} C_VEL
LIN {X 0,Y 277.651,Z 305.9,A -85,B 0,C 180,E1 -17542.727,E2 -17542.727} C_VEL
LIN {X 0,Y 277.819,Z 305.88,A -85,B 0,C 180,E1 -17548.548,E2 -17548.548} C_VEL
LIN {X 0,Y 277.819,Z 305.876,A -85,B 0,C 180,E1 -17551.447,E2 -17551.447} C_VEL
LIN {X 0,Y 277.648,Z 305.898,A -85,B 0,C 180,E1 -17557.268,E2 -17557.268} C_VEL
LIN {X 0,Y 277.501,Z 305.916,A -85,B 0,C 180,E1 -17560.208,E2 -17560.208} C_VEL
LIN {X 0,Y 277.427,Z 305.928,A -85,B 0,C 180,E1 -17564.671,E2 -17564.671} C_VEL
LIN {X 0,Y 277.364,Z 305.936,A -85,B 0,C 180,E1 -17569.228,E2 -17569.228} C_VEL
LIN {X 0,Y 277.318,Z 305.939,A -85,B 0,C 180,E1 -17573.916,E2 -17573.916} C_VEL
LIN {X 0,Y 277.314,Z 305.94,A -85,B 0,C 180,E1 -17577.502,E2 -17577.502} C_VEL
LIN {X 0,Y 277.256,Z 305.947,A -85,B 0,C 180,E1 -17580.477,E2 -17580.477} C_VEL
LIN {X 0,Y 277.236,Z 305.949,A -85,B 0,C 180,E1 -17583.891,E2 -17583.891} C_VEL
LIN {X 0,Y 277.285,Z 305.944,A -85,B 0,C 180,E1 -17585.801,E2 -17585.801} C_VEL
LIN {X 0,Y 285.508,Z 328.711,A -85,B 0,C 180,E1 -17587.139,E2 -17587.139} C_VEL
LIN {X 0,Y 287.526,Z 335.089,A -85,B 0,C 180,E1 -17587.475,E2 -17587.475} C_VEL
LIN {X 0,Y 284.78,Z 410.047,A -85,B 0,C 180,E1 -17589.792,E2 -17589.792} C_VEL
LIN {X 0,Y 284.225,Z 422.753,A -85,B 0,C 180,E1 -17590.438,E2 -17590.438} C_VEL
LIN {X 0,Y 283.358,Z 435.907,A -85,B 0,C 180,E1 -17591.387,E2 -17591.387} C_VEL
LIN {X 0,Y 282.263,Z 448.133,A -85,B 0,C 180,E1 -17592.575,E2 -17592.575} C_VEL
LIN {X 0,Y 280.987,Z 460.373,A -85,B 0,C 180,E1 -17594.104,E2 -17594.104} C_VEL
LIN {X 0,Y 279.842,Z 470.933,A -85,B 0,C 180,E1 -17595.78,E2 -17595.78} C_VEL
LIN {X 0,Y 278.588,Z 481.201,A -85,B 0,C 180,E1 -17597.805,E2 -17597.805} C_VEL
LIN {X 0,Y 277.679,Z 488.919,A -85,B 0,C 180,E1 -17599.686,E2 -17599.686} C_VEL
LIN {X 0,Y 276.824,Z 496.235,A -85,B 0,C 180,E1 -17601.897,E2 -17601.897} C_VEL
LIN {X 0,Y 276.189,Z 502.227,A -85,B 0,C 180,E1 -17604.179,E2 -17604.179} C_VEL
LIN {X 0,Y 275.769,Z 507.225,A -85,B 0,C 180,E1 -17606.654,E2 -17606.654} C_VEL
LIN {X 0,Y 275.356,Z 510.987,A -85,B 0,C 180,E1 -17609.306,E2 -17609.306} C_VEL
LIN {X 0,Y 275.285,Z 512.62,A -85,B 0,C 180,E1 -17610.984,E2 -17610.984} C_VEL
LIN {X 0,Y 275.341,Z 513.941,A -85,B 0,C 180,E1 -17613.282,E2 -17613.282} C_VEL
LIN {X 0,Y 275.697,Z 514.205,A -85,B 0,C 180,E1 -17615.93,E2 -17615.93} C_VEL
LIN {X 0,Y 276.078,Z 513.664,A -85,B 0,C 180,E1 -17617.553,E2 -17617.553} C_VEL
LIN {X 0,Y 276.866,Z 512.005,A -85,B 0,C 180,E1 -17619.897,E2 -17619.897} C_VEL
LIN {X 0,Y 277.914,Z 509.099,A -85,B 0,C 180,E1 -17622.335,E2 -17622.335} C_VEL
LIN {X 0,Y 279.299,Z 505.045,A -85,B 0,C 180,E1 -17624.681,E2 -17624.681} C_VEL
LIN {X 0,Y 281.129,Z 499.333,A -85,B 0,C 180,E1 -17627.118,E2 -17627.118} C_VEL
LIN {X 0,Y 283.107,Z 492.807,A -85,B 0,C 180,E1 -17629.271,E2 -17629.271} C_VEL
LIN {X 0,Y 285.013,Z 486.124,A -85,B 0,C 180,E1 -17631.047,E2 -17631.047} C_VEL
LIN {X 0,Y 287.36,Z 477.177,A -85,B 0,C 180,E1 -17632.977,E2 -17632.977} C_VEL
LIN {X 0,Y 289.458,Z 468.615,A -85,B 0,C 180,E1 -17634.463,E2 -17634.463} C_VEL
LIN {X 0,Y 291.73,Z 457.532,A -85,B 0,C 180,E1 -17636.029,E2 -17636.029} C_VEL
LIN {X 0,Y 293.46,Z 447.989,A -85,B 0,C 180,E1 -17637.116,E2 -17637.116} C_VEL
LIN {X 0,Y 293.815,Z 442.862,A -85,B 0,C 180,E1 -17637.686,E2 -17637.686} C_VEL
LIN {X 0,Y 292.792,Z 434.547,A -85,B 0,C 180,E1 -17638.72,E2 -17638.72} C_VEL
LIN {X 0,Y 291.544,Z 425.99,A -85,B 0,C 180,E1 -17639.657,E2 -17639.657} C_VEL
LIN {X 0,Y 291.466,Z 420.488,A -85,B 0,C 180,E1 -17640.068,E2 -17640.068} C_VEL
LIN {X 0,Y 292.466,Z 407.799,A -85,B 0,C 180,E1 -17640.603,E2 -17640.603} C_VEL
LIN {X 0,Y 296.43,Z 349.675,A -85,B 0,C 180,E1 -17642.517,E2 -17642.517} C_VEL
LIN {X 0,Y 292.927,Z 341.799,A -85,B 0,C 180,E1 -17643.542,E2 -17643.542} C_VEL
LIN {X 0,Y 289.082,Z 334.534,A -85,B 0,C 180,E1 -17644.705,E2 -17644.705} C_VEL
LIN {X 0,Y 282.788,Z 324.853,A -85,B 0,C 180,E1 -17646.671,E2 -17646.671} C_VEL
LIN {X 0,Y 277.872,Z 317.63,A -85,B 0,C 180,E1 -17648.368,E2 -17648.368} C_VEL
LIN {X 0,Y 272.976,Z 311.441,A -85,B 0,C 180,E1 -17650.22,E2 -17650.22} C_VEL
LIN {X 0,Y 271.071,Z 309.169,A -85,B 0,C 180,E1 -17651.001,E2 -17651.001} C_VEL
LIN {X 0,Y 270.806,Z 308.57,A -85,B 0,C 180,E1 -17651.225,E2 -17651.225} C_VEL
LIN {X 0,Y 270.324,Z 306.808,A -85,B 0,C 180,E1 -17652.386,E2 -17652.386} C_VEL
LIN {X 0,Y 270.295,Z 306.812,A -85,B 0,C 180,E1 -17655.865,E2 -17655.865} C_VEL
LIN {X 0,Y 270.208,Z 306.819,A -85,B 0,C 180,E1 -17660.576,E2 -17660.576} C_VEL
LIN {X 0,Y 270.203,Z 306.828,A -85,B 0,C 180,E1 -17664.593,E2 -17664.593} C_VEL
LIN {X 0,Y 270.212,Z 306.824,A -85,B 0,C 180,E1 -17667.916,E2 -17667.916} C_VEL
LIN {X 0,Y 270.144,Z 306.828,A -85,B 0,C 180,E1 -17671.354,E2 -17671.354} C_VEL
LIN {X 0,Y 270.175,Z 306.824,A -85,B 0,C 180,E1 -17674.91,E2 -17674.91} C_VEL
LIN {X 0,Y 270.199,Z 306.828,A -85,B 0,C 180,E1 -17678.722,E2 -17678.722} C_VEL
LIN {X 0,Y 270.182,Z 306.985,A -85,B 0,C 180,E1 -17683.127,E2 -17683.127} C_VEL
LIN {X 0,Y 272.677,Z 313.643,A -85,B 0,C 180,E1 -17687.336,E2 -17687.336} C_VEL
LIN {X 0,Y 274.572,Z 319.155,A -85,B 0,C 180,E1 -17690.223,E2 -17690.223} C_VEL
LIN {X 0,Y 276.283,Z 324.521,A -85,B 0,C 180,E1 -17692.648,E2 -17692.648} C_VEL
LIN {X 0,Y 280.337,Z 331.597,A -85,B 0,C 180,E1 -17694.144,E2 -17694.144} C_VEL
LIN {X 0,Y 283.879,Z 338.168,A -85,B 0,C 180,E1 -17695.378,E2 -17695.378} C_VEL
LIN {X 0,Y 286.88,Z 344.213,A -85,B 0,C 180,E1 -17696.356,E2 -17696.356} C_VEL
LIN {X 0,Y 290.366,Z 352.174,A -85,B 0,C 180,E1 -17697.491,E2 -17697.491} C_VEL
LIN {X 0,Y 291.912,Z 360.741,A -85,B 0,C 180,E1 -17698.202,E2 -17698.202} C_VEL
LIN {X 0,Y 293.736,Z 375.203,A -85,B 0,C 180,E1 -17699.208,E2 -17699.208} C_VEL
LIN {X 0,Y 294.508,Z 385.971,A -85,B 0,C 180,E1 -17699.831,E2 -17699.831} C_VEL
LIN {X 0,Y 290.846,Z 439.272,A -85,B 0,C 180,E1 -17701.599,E2 -17701.599} C_VEL
LIN {X 0,Y 289.172,Z 453.155,A -85,B 0,C 180,E1 -17702.308,E2 -17702.308} C_VEL
LIN {X 0,Y 286.922,Z 466.244,A -85,B 0,C 180,E1 -17703.256,E2 -17703.256} C_VEL
LIN {X 0,Y 284.534,Z 478.009,A -85,B 0,C 180,E1 -17704.395,E2 -17704.395} C_VEL
LIN {X 0,Y 282.114,Z 488.787,A -85,B 0,C 180,E1 -17705.735,E2 -17705.735} C_VEL
LIN {X 0,Y 279.342,Z 499.669,A -85,B 0,C 180,E1 -17707.443,E2 -17707.443} C_VEL
LIN {X 0,Y 276.944,Z 508.684,A -85,B 0,C 180,E1 -17709.194,E2 -17709.194} C_VEL
LIN {X 0,Y 274.773,Z 516.313,A -85,B 0,C 180,E1 -17711,E2 -17711} C_VEL
LIN {X 0,Y 272.831,Z 523.676,A -85,B 0,C 180,E1 -17713.159,E2 -17713.159} C_VEL
LIN {X 0,Y 271.363,Z 528.776,A -85,B 0,C 180,E1 -17714.994,E2 -17714.994} C_VEL
LIN {X 0,Y 269.896,Z 533.79,A -85,B 0,C 180,E1 -17717.216,E2 -17717.216} C_VEL
LIN {X 0,Y 269.021,Z 537.709,A -85,B 0,C 180,E1 -17719.467,E2 -17719.467} C_VEL
LIN {X 0,Y 268.655,Z 539.771,A -85,B 0,C 180,E1 -17720.973,E2 -17720.973} C_VEL
LIN {X 0,Y 268.373,Z 541.356,A -85,B 0,C 180,E1 -17722.479,E2 -17722.479} C_VEL
LIN {X 0,Y 268.248,Z 542.927,A -85,B 0,C 180,E1 -17724.621,E2 -17724.621} C_VEL
LIN {X 0,Y 268.326,Z 543.67,A -85,B 0,C 180,E1 -17727,E2 -17727} C_VEL
LIN {X 0,Y 268.366,Z 543.577,A -85,B 0,C 180,E1 -17728.502,E2 -17728.502} C_VEL
LIN {X 0,Y 268.582,Z 543.073,A -85,B 0,C 180,E1 -17730.002,E2 -17730.002} C_VEL
LIN {X 0,Y 268.452,Z 542.122,A -85,B 0,C 180,E1 -17731.502,E2 -17731.502} C_VEL
LIN {X 0,Y 268.403,Z 540.728,A -85,B 0,C 180,E1 -17733.004,E2 -17733.004} C_VEL
LIN {X 0,Y 268.482,Z 537.654,A -85,B 0,C 180,E1 -17735.31,E2 -17735.31} C_VEL
LIN {X 0,Y 268.526,Z 533.585,A -85,B 0,C 180,E1 -17737.521,E2 -17737.521} C_VEL
LIN {X 0,Y 268.883,Z 527.128,A -85,B 0,C 180,E1 -17740.163,E2 -17740.163} C_VEL
LIN {X 0,Y 269.537,Z 520.051,A -85,B 0,C 180,E1 -17742.423,E2 -17742.423} C_VEL
LIN {X 0,Y 270.507,Z 511.125,A -85,B 0,C 180,E1 -17744.675,E2 -17744.675} C_VEL
LIN {X 0,Y 271.329,Z 503.948,A -85,B 0,C 180,E1 -17746.168,E2 -17746.168} C_VEL
LIN {X 0,Y 272.763,Z 493.129,A -85,B 0,C 180,E1 -17748.011,E2 -17748.011} C_VEL
LIN {X 0,Y 274.002,Z 482.385,A -85,B 0,C 180,E1 -17749.478,E2 -17749.478} C_VEL
LIN {X 0,Y 275.218,Z 470.467,A -85,B 0,C 180,E1 -17750.752,E2 -17750.752} C_VEL
LIN {X 0,Y 276.524,Z 457.181,A -85,B 0,C 180,E1 -17751.821,E2 -17751.821} C_VEL
LIN {X 0,Y 277.528,Z 443.636,A -85,B 0,C 180,E1 -17752.57,E2 -17752.57} C_VEL
LIN {X 0,Y 278.3,Z 422.785,A -85,B 0,C 180,E1 -17753.289,E2 -17753.289} C_VEL
LIN {X 0,Y 279.592,Z 380.026,A -85,B 0,C 180,E1 -17754.657,E2 -17754.657} C_VEL
LIN {X 0,Y 274.37,Z 332.491,A -85,B 0,C 180,E1 -17756.654,E2 -17756.654} C_VEL
LIN {X 0,Y 274.596,Z 328.404,A -85,B 0,C 180,E1 -17757.845,E2 -17757.845} C_VEL
LIN {X 0,Y 272.245,Z 316.492,A -85,B 0,C 180,E1 -17761.58,E2 -17761.58} C_VEL
LIN {X 0,Y 270.241,Z 306.823,A -85,B 0,C 180,E1 -17764.75,E2 -17764.75} C_VEL
LIN {X 0,Y 270.166,Z 306.833,A -85,B 0,C 180,E1 -17768.701,E2 -17768.701} C_VEL
LIN {X 0,Y 270.142,Z 306.834,A -85,B 0,C 180,E1 -17773.243,E2 -17773.243} C_VEL
LIN {X 0,Y 270.141,Z 306.833,A -85,B 0,C 180,E1 -17777.435,E2 -17777.435} C_VEL
LIN {X 0,Y 270.169,Z 306.83,A -85,B 0,C 180,E1 -17781.367,E2 -17781.367} C_VEL
LIN {X 0,Y 270.184,Z 306.831,A -85,B 0,C 180,E1 -17785.091,E2 -17785.091} C_VEL
LIN {X 0,Y 270.173,Z 306.833,A -85,B 0,C 180,E1 -17789.135,E2 -17789.135} C_VEL
LIN {X 0,Y 270.213,Z 306.823,A -85,B 0,C 180,E1 -17792.161,E2 -17792.161} C_VEL
LIN {X 0,Y 270.215,Z 306.824,A -85,B 0,C 180,E1 -17795.541,E2 -17795.541} C_VEL
LIN {X 0,Y 270.208,Z 306.824,A -85,B 0,C 180,E1 -17800.237,E2 -17800.237} C_VEL
LIN {X 0,Y 270.351,Z 306.807,A -85,B 0,C 180,E1 -17804.932,E2 -17804.932} C_VEL
LIN {X 0,Y 270.371,Z 306.807,A -85,B 0,C 180,E1 -17809.515,E2 -17809.515} C_VEL
LIN {X 0,Y 270.572,Z 306.778,A -85,B 0,C 180,E1 -17812.537,E2 -17812.537} C_VEL
LIN {X 0,Y 270.763,Z 306.755,A -85,B 0,C 180,E1 -17818.512,E2 -17818.512} C_VEL
LIN {X 0,Y 270.763,Z 306.758,A -85,B 0,C 180,E1 -17821.487,E2 -17821.487} C_VEL
LIN {X 0,Y 270.567,Z 306.783,A -85,B 0,C 180,E1 -17827.462,E2 -17827.462} C_VEL
LIN {X 0,Y 270.394,Z 306.799,A -85,B 0,C 180,E1 -17830.482,E2 -17830.482} C_VEL
LIN {X 0,Y 270.35,Z 306.807,A -85,B 0,C 180,E1 -17835.067,E2 -17835.067} C_VEL
LIN {X 0,Y 270.205,Z 306.828,A -85,B 0,C 180,E1 -17839.762,E2 -17839.762} C_VEL
LIN {X 0,Y 270.223,Z 306.822,A -85,B 0,C 180,E1 -17844.59,E2 -17844.59} C_VEL
LIN {X 0,Y 270.257,Z 306.821,A -85,B 0,C 180,E1 -17847.909,E2 -17847.909} C_VEL
LIN {X 0,Y 270.171,Z 306.83,A -85,B 0,C 180,E1 -17851.349,E2 -17851.349} C_VEL
LIN {X 0,Y 270.189,Z 306.825,A -85,B 0,C 180,E1 -17854.906,E2 -17854.906} C_VEL
LIN {X 0,Y 270.187,Z 306.827,A -85,B 0,C 180,E1 -17858.711,E2 -17858.711} C_VEL
LIN {X 0,Y 270.163,Z 306.829,A -85,B 0,C 180,E1 -17863.251,E2 -17863.251} C_VEL
LIN {X 0,Y 270.205,Z 306.825,A -85,B 0,C 180,E1 -17867.45,E2 -17867.45} C_VEL
LIN {X 0,Y 270.239,Z 306.82,A -85,B 0,C 180,E1 -17871.381,E2 -17871.381} C_VEL
LIN {X 0,Y 270.21,Z 306.823,A -85,B 0,C 180,E1 -17875.097,E2 -17875.097} C_VEL
LIN {X 0,Y 270.196,Z 306.825,A -85,B 0,C 180,E1 -17879.131,E2 -17879.131} C_VEL
LIN {X 0,Y 270.259,Z 306.82,A -85,B 0,C 180,E1 -17882.146,E2 -17882.146} C_VEL
LIN {X 0,Y 270.274,Z 306.816,A -85,B 0,C 180,E1 -17885.519,E2 -17885.519} C_VEL
LIN {X 0,Y 270.3,Z 306.815,A -85,B 0,C 180,E1 -17890.244,E2 -17890.244} C_VEL
LIN {X 0,Y 270.401,Z 306.801,A -85,B 0,C 180,E1 -17894.934,E2 -17894.934} C_VEL
LIN {X 0,Y 270.44,Z 306.794,A -85,B 0,C 180,E1 -17899.518,E2 -17899.518} C_VEL
LIN {X 0,Y 270.609,Z 306.779,A -85,B 0,C 180,E1 -17902.537,E2 -17902.537} C_VEL
LIN {X 0,Y 270.785,Z 306.755,A -85,B 0,C 180,E1 -17908.511,E2 -17908.511} C_VEL
LIN {X 0,Y 270.785,Z 306.752,A -85,B 0,C 180,E1 -17911.485,E2 -17911.485} C_VEL
LIN {X 0,Y 270.606,Z 306.775,A -85,B 0,C 180,E1 -17917.458,E2 -17917.458} C_VEL
LIN {X 0,Y 270.436,Z 306.798,A -85,B 0,C 180,E1 -17920.478,E2 -17920.478} C_VEL
LIN {X 0,Y 270.396,Z 306.803,A -85,B 0,C 180,E1 -17925.061,E2 -17925.061} C_VEL
LIN {X 0,Y 270.318,Z 306.811,A -85,B 0,C 180,E1 -17929.75,E2 -17929.75} C_VEL
LIN {X 0,Y 270.262,Z 306.82,A -85,B 0,C 180,E1 -17934.581,E2 -17934.581} C_VEL
LIN {X 0,Y 270.258,Z 306.818,A -85,B 0,C 180,E1 -17937.904,E2 -17937.904} C_VEL
LIN {X 0,Y 270.168,Z 306.832,A -85,B 0,C 180,E1 -17941.344,E2 -17941.344} C_VEL
LIN {X 0,Y 270.222,Z 306.827,A -85,B 0,C 180,E1 -17945.294,E2 -17945.294} C_VEL
LIN {X 0,Y 272.73,Z 313.736,A -85,B 0,C 180,E1 -17945.759,E2 -17945.759} C_VEL
LIN {X 0,Y 279.154,Z 331.387,A -85,B 0,C 180,E1 -17946.818,E2 -17946.818} C_VEL
LIN {X 0,Y 280.656,Z 336.223,A -85,B 0,C 180,E1 -17947.08,E2 -17947.08} C_VEL
LIN {X 0,Y 277.851,Z 411.336,A -85,B 0,C 180,E1 -17949.482,E2 -17949.482} C_VEL
LIN {X 0,Y 277.271,Z 424.929,A -85,B 0,C 180,E1 -17950.221,E2 -17950.221} C_VEL
LIN {X 0,Y 276.321,Z 437.39,A -85,B 0,C 180,E1 -17951.175,E2 -17951.175} C_VEL
LIN {X 0,Y 275.188,Z 450.002,A -85,B 0,C 180,E1 -17952.467,E2 -17952.467} C_VEL
LIN {X 0,Y 274.034,Z 460.434,A -85,B 0,C 180,E1 -17953.816,E2 -17953.816} C_VEL
LIN {X 0,Y 272.923,Z 470.551,A -85,B 0,C 180,E1 -17955.437,E2 -17955.437} C_VEL
LIN {X 0,Y 271.637,Z 480.787,A -85,B 0,C 180,E1 -17957.475,E2 -17957.475} C_VEL
LIN {X 0,Y 270.638,Z 489.09,A -85,B 0,C 180,E1 -17959.519,E2 -17959.519} C_VEL
LIN {X 0,Y 269.757,Z 496.511,A -85,B 0,C 180,E1 -17961.803,E2 -17961.803} C_VEL
LIN {X 0,Y 269.136,Z 502.29,A -85,B 0,C 180,E1 -17964.036,E2 -17964.036} C_VEL
LIN {X 0,Y 268.674,Z 507.549,A -85,B 0,C 180,E1 -17966.681,E2 -17966.681} C_VEL
LIN {X 0,Y 268.397,Z 510.139,A -85,B 0,C 180,E1 -17968.42,E2 -17968.42} C_VEL
LIN {X 0,Y 268.214,Z 512.136,A -85,B 0,C 180,E1 -17970.143,E2 -17970.143} C_VEL
LIN {X 0,Y 268.227,Z 514.133,A -85,B 0,C 180,E1 -17972.964,E2 -17972.964} C_VEL
LIN {X 0,Y 268.505,Z 514.69,A -85,B 0,C 180,E1 -17975.242,E2 -17975.242} C_VEL
LIN {X 0,Y 268.858,Z 514.476,A -85,B 0,C 180,E1 -17976.915,E2 -17976.915} C_VEL
LIN {X 0,Y 269.704,Z 513.005,A -85,B 0,C 180,E1 -17979.711,E2 -17979.711} C_VEL
LIN {X 0,Y 271.013,Z 509.794,A -85,B 0,C 180,E1 -17982.651,E2 -17982.651} C_VEL
LIN {X 0,Y 272.461,Z 505.863,A -85,B 0,C 180,E1 -17985.053,E2 -17985.053} C_VEL
LIN {X 0,Y 274.491,Z 500.094,A -85,B 0,C 180,E1 -17987.628,E2 -17987.628} C_VEL
LIN {X 0,Y 276.825,Z 492.808,A -85,B 0,C 180,E1 -17990.074,E2 -17990.074} C_VEL
LIN {X 0,Y 279.064,Z 485.379,A -85,B 0,C 180,E1 -17992.039,E2 -17992.039} C_VEL
LIN {X 0,Y 281.514,Z 476.637,A -85,B 0,C 180,E1 -17993.91,E2 -17993.91} C_VEL
LIN {X 0,Y 284.188,Z 465.827,A -85,B 0,C 180,E1 -17995.746,E2 -17995.746} C_VEL
LIN {X 0,Y 286.453,Z 455.181,A -85,B 0,C 180,E1 -17997.188,E2 -17997.188} C_VEL
LIN {X 0,Y 288.521,Z 443.48,A -85,B 0,C 180,E1 -17998.428,E2 -17998.428} C_VEL
LIN {X 0,Y 290.442,Z 430.299,A -85,B 0,C 180,E1 -17999.481,E2 -17999.481} C_VEL
LIN {X 0,Y 291.466,Z 420.488,A -85,B 0,C 180,E1 -18000.068,E2 -18000.068} C_VEL
LIN {X 0,Y 291.428,Z 414.881,A -85,B 0,C 180,E1 -18000.436,E2 -18000.436} C_VEL
LIN {X 0,Y 288.484,Z 396.597,A -85,B 0,C 180,E1 -18001.816,E2 -18001.816} C_VEL
LIN {X 0,Y 288.296,Z 390.876,A -85,B 0,C 180,E1 -18002.105,E2 -18002.105} C_VEL
LIN {X 0,Y 291.106,Z 352.148,A -85,B 0,C 180,E1 -18003.403,E2 -18003.403} C_VEL
LIN {X 0,Y 288.081,Z 345.248,A -85,B 0,C 180,E1 -18004.373,E2 -18004.373} C_VEL
LIN {X 0,Y 284.626,Z 338.835,A -85,B 0,C 180,E1 -18005.458,E2 -18005.458} C_VEL
LIN {X 0,Y 278.842,Z 329.764,A -85,B 0,C 180,E1 -18007.388,E2 -18007.388} C_VEL
LIN {X 0,Y 275.708,Z 324.966,A -85,B 0,C 180,E1 -18008.526,E2 -18008.526} C_VEL
LIN {X 0,Y 273.204,Z 321.603,A -85,B 0,C 180,E1 -18009.48,E2 -18009.48} C_VEL
LIN {X 0,Y 270.365,Z 317.76,A -85,B 0,C 180,E1 -18010.627,E2 -18010.627} C_VEL
LIN {X 0,Y 268.117,Z 314.978,A -85,B 0,C 180,E1 -18011.602,E2 -18011.602} C_VEL
LIN {X 0,Y 264.031,Z 310.074,A -85,B 0,C 180,E1 -18013.538,E2 -18013.538} C_VEL
LIN {X 0,Y 263.273,Z 307.685,A -85,B 0,C 180,E1 -18015.483,E2 -18015.483} C_VEL
LIN {X 0,Y 263.174,Z 307.694,A -85,B 0,C 180,E1 -18020.315,E2 -18020.315} C_VEL
LIN {X 0,Y 263.156,Z 307.7,A -85,B 0,C 180,E1 -18025.297,E2 -18025.297} C_VEL
LIN {X 0,Y 263.123,Z 307.702,A -85,B 0,C 180,E1 -18028.737,E2 -18028.737} C_VEL
LIN {X 0,Y 263.099,Z 307.706,A -85,B 0,C 180,E1 -18032.294,E2 -18032.294} C_VEL
LIN {X 0,Y 263.169,Z 307.698,A -85,B 0,C 180,E1 -18036.771,E2 -18036.771} C_VEL
LIN {X 0,Y 263.124,Z 307.755,A -85,B 0,C 180,E1 -18040.114,E2 -18040.114} C_VEL
LIN {X 0,Y 264.76,Z 312.18,A -85,B 0,C 180,E1 -18043.644,E2 -18043.644} C_VEL
LIN {X 0,Y 266.994,Z 318.139,A -85,B 0,C 180,E1 -18047.48,E2 -18047.48} C_VEL
LIN {X 0,Y 268.826,Z 323.518,A -85,B 0,C 180,E1 -18050.299,E2 -18050.299} C_VEL
LIN {X 0,Y 273.461,Z 331.18,A -85,B 0,C 180,E1 -18052.258,E2 -18052.258} C_VEL
LIN {X 0,Y 276.815,Z 337.079,A -85,B 0,C 180,E1 -18053.553,E2 -18053.553} C_VEL
LIN {X 0,Y 280.021,Z 343.186,A -85,B 0,C 180,E1 -18054.719,E2 -18054.719} C_VEL
LIN {X 0,Y 283.8,Z 351.221,A -85,B 0,C 180,E1 -18056.043,E2 -18056.043} C_VEL
LIN {X 0,Y 286.019,Z 356.975,A -85,B 0,C 180,E1 -18056.822,E2 -18056.822} C_VEL
LIN {X 0,Y 288.154,Z 373.24,A -85,B 0,C 180,E1 -18058.08,E2 -18058.08} C_VEL
LIN {X 0,Y 289.254,Z 386.174,A -85,B 0,C 180,E1 -18058.893,E2 -18058.893} C_VEL
LIN {X 0,Y 285.462,Z 438.341,A -85,B 0,C 180,E1 -18060.66,E2 -18060.66} C_VEL
LIN {X 0,Y 283.611,Z 452.842,A -85,B 0,C 180,E1 -18061.414,E2 -18061.414} C_VEL
LIN {X 0,Y 281.443,Z 464.84,A -85,B 0,C 180,E1 -18062.29,E2 -18062.29} C_VEL
LIN {X 0,Y 278.587,Z 478.307,A -85,B 0,C 180,E1 -18063.606,E2 -18063.606} C_VEL
LIN {X 0,Y 275.748,Z 490.086,A -85,B 0,C 180,E1 -18065.137,E2 -18065.137} C_VEL
LIN {X 0,Y 272.871,Z 500.695,A -85,B 0,C 180,E1 -18066.878,E2 -18066.878} C_VEL
LIN {X 0,Y 270.374,Z 509.418,A -85,B 0,C 180,E1 -18068.664,E2 -18068.664} C_VEL
LIN {X 0,Y 268.036,Z 516.984,A -85,B 0,C 180,E1 -18070.557,E2 -18070.557} C_VEL
LIN {X 0,Y 266.039,Z 523.967,A -85,B 0,C 180,E1 -18072.715,E2 -18072.715} C_VEL
LIN {X 0,Y 263.961,Z 530.715,A -85,B 0,C 180,E1 -18075.353,E2 -18075.353} C_VEL
LIN {X 0,Y 262.561,Z 535.217,A -85,B 0,C 180,E1 -18077.639,E2 -18077.639} C_VEL
LIN {X 0,Y 262.006,Z 537.64,A -85,B 0,C 180,E1 -18079.181,E2 -18079.181} C_VEL
LIN {X 0,Y 261.596,Z 539.591,A -85,B 0,C 180,E1 -18080.727,E2 -18080.727} C_VEL
LIN {X 0,Y 261.223,Z 542.241,A -85,B 0,C 180,E1 -18083.825,E2 -18083.825} C_VEL
LIN {X 0,Y 261.156,Z 542.961,A -85,B 0,C 180,E1 -18085.372,E2 -18085.372} C_VEL
LIN {X 0,Y 261.252,Z 543.237,A -85,B 0,C 180,E1 -18086.919,E2 -18086.919} C_VEL
LIN {X 0,Y 261.497,Z 542.53,A -85,B 0,C 180,E1 -18090.002,E2 -18090.002} C_VEL
LIN {X 0,Y 261.367,Z 541.527,A -85,B 0,C 180,E1 -18091.543,E2 -18091.543} C_VEL
LIN {X 0,Y 261.337,Z 540.039,A -85,B 0,C 180,E1 -18093.085,E2 -18093.085} C_VEL
LIN {X 0,Y 261.416,Z 538.1,A -85,B 0,C 180,E1 -18094.628,E2 -18094.628} C_VEL
LIN {X 0,Y 261.426,Z 534.238,A -85,B 0,C 180,E1 -18096.95,E2 -18096.95} C_VEL
LIN {X 0,Y 261.631,Z 529.15,A -85,B 0,C 180,E1 -18099.277,E2 -18099.277} C_VEL
LIN {X 0,Y 262.122,Z 522.681,A -85,B 0,C 180,E1 -18101.602,E2 -18101.602} C_VEL
LIN {X 0,Y 263.054,Z 514.527,A -85,B 0,C 180,E1 -18103.914,E2 -18103.914} C_VEL
LIN {X 0,Y 264.1,Z 506.193,A -85,B 0,C 180,E1 -18105.83,E2 -18105.83} C_VEL
LIN {X 0,Y 265.26,Z 496.449,A -85,B 0,C 180,E1 -18107.661,E2 -18107.661} C_VEL
LIN {X 0,Y 266.568,Z 485.964,A -85,B 0,C 180,E1 -18109.243,E2 -18109.243} C_VEL
LIN {X 0,Y 267.983,Z 473.397,A -85,B 0,C 180,E1 -18110.735,E2 -18110.735} C_VEL
LIN {X 0,Y 269.234,Z 461.177,A -85,B 0,C 180,E1 -18111.838,E2 -18111.838} C_VEL
LIN {X 0,Y 270.371,Z 447.083,A -85,B 0,C 180,E1 -18112.747,E2 -18112.747} C_VEL
LIN {X 0,Y 270.975,Z 433.931,A -85,B 0,C 180,E1 -18113.299,E2 -18113.299} C_VEL
LIN {X 0,Y 272.841,Z 381.802,A -85,B 0,C 180,E1 -18114.997,E2 -18114.997} C_VEL
LIN {X 0,Y 267.494,Z 332.149,A -85,B 0,C 180,E1 -18117.135,E2 -18117.135} C_VEL
LIN {X 0,Y 267.435,Z 328.555,A -85,B 0,C 180,E1 -18118.231,E2 -18118.231} C_VEL
LIN {X 0,Y 265.074,Z 316.823,A -85,B 0,C 180,E1 -18122.023,E2 -18122.023} C_VEL
LIN {X 0,Y 263.183,Z 307.701,A -85,B 0,C 180,E1 -18125.167,E2 -18125.167} C_VEL
LIN {X 0,Y 263.088,Z 307.712,A -85,B 0,C 180,E1 -18129.222,E2 -18129.222} C_VEL
LIN {X 0,Y 263.07,Z 307.713,A -85,B 0,C 180,E1 -18131.902,E2 -18131.902} C_VEL
LIN {X 0,Y 263.072,Z 307.712,A -85,B 0,C 180,E1 -18136.16,E2 -18136.16} C_VEL
LIN {X 0,Y 263.106,Z 307.712,A -85,B 0,C 180,E1 -18140.769,E2 -18140.769} C_VEL
LIN {X 0,Y 263.145,Z 307.704,A -85,B 0,C 180,E1 -18144.014,E2 -18144.014} C_VEL
LIN {X 0,Y 263.11,Z 307.709,A -85,B 0,C 180,E1 -18147.708,E2 -18147.708} C_VEL
LIN {X 0,Y 263.138,Z 307.705,A -85,B 0,C 180,E1 -18151.803,E2 -18151.803} C_VEL
LIN {X 0,Y 263.178,Z 307.703,A -85,B 0,C 180,E1 -18155.217,E2 -18155.217} C_VEL
LIN {X 0,Y 263.195,Z 307.699,A -85,B 0,C 180,E1 -18159.687,E2 -18159.687} C_VEL
LIN {X 0,Y 263.294,Z 307.684,A -85,B 0,C 180,E1 -18164.518,E2 -18164.518} C_VEL
LIN {X 0,Y 263.317,Z 307.686,A -85,B 0,C 180,E1 -18169.231,E2 -18169.231} C_VEL
LIN {X 0,Y 263.534,Z 307.654,A -85,B 0,C 180,E1 -18172.337,E2 -18172.337} C_VEL
LIN {X 0,Y 263.728,Z 307.631,A -85,B 0,C 180,E1 -18178.472,E2 -18178.472} C_VEL
LIN {X 0,Y 263.728,Z 307.634,A -85,B 0,C 180,E1 -18181.526,E2 -18181.526} C_VEL
LIN {X 0,Y 263.53,Z 307.66,A -85,B 0,C 180,E1 -18187.662,E2 -18187.662} C_VEL
LIN {X 0,Y 263.333,Z 307.678,A -85,B 0,C 180,E1 -18190.766,E2 -18190.766} C_VEL
LIN {X 0,Y 263.292,Z 307.689,A -85,B 0,C 180,E1 -18195.481,E2 -18195.481} C_VEL
LIN {X 0,Y 263.192,Z 307.698,A -85,B 0,C 180,E1 -18200.311,E2 -18200.311} C_VEL
LIN {X 0,Y 263.178,Z 307.701,A -85,B 0,C 180,E1 -18205.294,E2 -18205.294} C_VEL
LIN {X 0,Y 263.153,Z 307.702,A -85,B 0,C 180,E1 -18208.732,E2 -18208.732} C_VEL
LIN {X 0,Y 263.12,Z 307.709,A -85,B 0,C 180,E1 -18212.289,E2 -18212.289} C_VEL
LIN {X 0,Y 263.181,Z 307.698,A -85,B 0,C 180,E1 -18216.766,E2 -18216.766} C_VEL
LIN {X 0,Y 263.117,Z 307.709,A -85,B 0,C 180,E1 -18221.594,E2 -18221.594} C_VEL
LIN {X 0,Y 263.131,Z 307.709,A -85,B 0,C 180,E1 -18226.02,E2 -18226.02} C_VEL
LIN {X 0,Y 263.152,Z 307.707,A -85,B 0,C 180,E1 -18230.138,E2 -18230.138} C_VEL
LIN {X 0,Y 263.184,Z 307.701,A -85,B 0,C 180,E1 -18234.023,E2 -18234.023} C_VEL
LIN {X 0,Y 263.128,Z 307.707,A -85,B 0,C 180,E1 -18237.712,E2 -18237.712} C_VEL
LIN {X 0,Y 263.192,Z 307.697,A -85,B 0,C 180,E1 -18241.785,E2 -18241.785} C_VEL
LIN {X 0,Y 263.223,Z 307.694,A -85,B 0,C 180,E1 -18245.2,E2 -18245.2} C_VEL
LIN {X 0,Y 263.262,Z 307.688,A -85,B 0,C 180,E1 -18249.693,E2 -18249.693} C_VEL
LIN {X 0,Y 263.349,Z 307.682,A -85,B 0,C 180,E1 -18254.521,E2 -18254.521} C_VEL
LIN {X 0,Y 263.372,Z 307.675,A -85,B 0,C 180,E1 -18259.233,E2 -18259.233} C_VEL
LIN {X 0,Y 263.571,Z 307.654,A -85,B 0,C 180,E1 -18262.337,E2 -18262.337} C_VEL
LIN {X 0,Y 263.749,Z 307.631,A -85,B 0,C 180,E1 -18268.471,E2 -18268.471} C_VEL
LIN {X 0,Y 263.749,Z 307.629,A -85,B 0,C 180,E1 -18271.524,E2 -18271.524} C_VEL
LIN {X 0,Y 263.568,Z 307.651,A -85,B 0,C 180,E1 -18277.658,E2 -18277.658} C_VEL
LIN {X 0,Y 263.369,Z 307.68,A -85,B 0,C 180,E1 -18280.762,E2 -18280.762} C_VEL
LIN {X 0,Y 263.344,Z 307.679,A -85,B 0,C 180,E1 -18285.474,E2 -18285.474} C_VEL
LIN {X 0,Y 263.278,Z 307.689,A -85,B 0,C 180,E1 -18290.301,E2 -18290.301} C_VEL
LIN {X 0,Y 263.197,Z 307.7,A -85,B 0,C 180,E1 -18295.287,E2 -18295.287} C_VEL
LIN {X 0,Y 263.165,Z 307.704,A -85,B 0,C 180,E1 -18298.725,E2 -18298.725} C_VEL
LIN {X 0,Y 263.116,Z 307.708,A -85,B 0,C 180,E1 -18302.284,E2 -18302.284} C_VEL
LIN {X 0,Y 263.149,Z 307.707,A -85,B 0,C 180,E1 -18304.828,E2 -18304.828} C_VEL
LIN {X 0,Y 272.484,Z 333.146,A -85,B 0,C 180,E1 -18306.428,E2 -18306.428} C_VEL
LIN {X 0,Y 273.858,Z 337.377,A -85,B 0,C 180,E1 -18306.669,E2 -18306.669} C_VEL
LIN {X 0,Y 270.993,Z 412.054,A -85,B 0,C 180,E1 -18309.134,E2 -18309.134} C_VEL
LIN {X 0,Y 270.376,Z 425.526,A -85,B 0,C 180,E1 -18309.89,E2 -18309.89} C_VEL
LIN {X 0,Y 269.405,Z 437.67,A -85,B 0,C 180,E1 -18310.842,E2 -18310.842} C_VEL
LIN {X 0,Y 268.176,Z 450.932,A -85,B 0,C 180,E1 -18312.241,E2 -18312.241} C_VEL
LIN {X 0,Y 266.814,Z 462.769,A -85,B 0,C 180,E1 -18313.858,E2 -18313.858} C_VEL
LIN {X 0,Y 265.549,Z 473.67,A -85,B 0,C 180,E1 -18315.742,E2 -18315.742} C_VEL
LIN {X 0,Y 264.349,Z 483.385,A -85,B 0,C 180,E1 -18317.838,E2 -18317.838} C_VEL
LIN {X 0,Y 263.27,Z 491.98,A -85,B 0,C 180,E1 -18320.158,E2 -18320.158} C_VEL
LIN {X 0,Y 262.463,Z 498.697,A -85,B 0,C 180,E1 -18322.417,E2 -18322.417} C_VEL
LIN {X 0,Y 261.899,Z 504.224,A -85,B 0,C 180,E1 -18324.765,E2 -18324.765} C_VEL
LIN {X 0,Y 261.426,Z 509.032,A -85,B 0,C 180,E1 -18327.476,E2 -18327.476} C_VEL
LIN {X 0,Y 261.195,Z 511.6,A -85,B 0,C 180,E1 -18329.417,E2 -18329.417} C_VEL
LIN {X 0,Y 261.098,Z 513.148,A -85,B 0,C 180,E1 -18331.021,E2 -18331.021} C_VEL
LIN {X 0,Y 261.141,Z 514.358,A -85,B 0,C 180,E1 -18332.774,E2 -18332.774} C_VEL
LIN {X 0,Y 261.291,Z 514.982,A -85,B 0,C 180,E1 -18334.511,E2 -18334.511} C_VEL
LIN {X 0,Y 261.595,Z 515.106,A -85,B 0,C 180,E1 -18336.236,E2 -18336.236} C_VEL
LIN {X 0,Y 262.018,Z 514.72,A -85,B 0,C 180,E1 -18337.945,E2 -18337.945} C_VEL
LIN {X 0,Y 262.605,Z 513.809,A -85,B 0,C 180,E1 -18339.641,E2 -18339.641} C_VEL
LIN {X 0,Y 263.29,Z 512.446,A -85,B 0,C 180,E1 -18341.319,E2 -18341.319} C_VEL
LIN {X 0,Y 264.648,Z 509.238,A -85,B 0,C 180,E1 -18343.918,E2 -18343.918} C_VEL
LIN {X 0,Y 266.255,Z 505.141,A -85,B 0,C 180,E1 -18346.258,E2 -18346.258} C_VEL
LIN {X 0,Y 268.34,Z 499.511,A -85,B 0,C 180,E1 -18348.673,E2 -18348.673} C_VEL
LIN {X 0,Y 270.759,Z 492.448,A -85,B 0,C 180,E1 -18351.041,E2 -18351.041} C_VEL
LIN {X 0,Y 273.121,Z 485.127,A -85,B 0,C 180,E1 -18352.98,E2 -18352.98} C_VEL
LIN {X 0,Y 275.684,Z 476.383,A -85,B 0,C 180,E1 -18354.842,E2 -18354.842} C_VEL
LIN {X 0,Y 278.285,Z 466.35,A -85,B 0,C 180,E1 -18356.562,E2 -18356.562} C_VEL
LIN {X 0,Y 280.872,Z 454.861,A -85,B 0,C 180,E1 -18358.124,E2 -18358.124} C_VEL
LIN {X 0,Y 283.236,Z 442.134,A -85,B 0,C 180,E1 -18359.468,E2 -18359.468} C_VEL
LIN {X 0,Y 285.08,Z 429.788,A -85,B 0,C 180,E1 -18360.442,E2 -18360.442} C_VEL
LIN {X 0,Y 286.359,Z 417.628,A -85,B 0,C 180,E1 -18361.143,E2 -18361.143} C_VEL
LIN {X 0,Y 288.057,Z 394.519,A -85,B 0,C 180,E1 -18361.979,E2 -18361.979} C_VEL
LIN {X 0,Y 288.296,Z 390.876,A -85,B 0,C 180,E1 -18362.105,E2 -18362.105} C_VEL
LIN {X 0,Y 288.139,Z 385.154,A -85,B 0,C 180,E1 -18362.404,E2 -18362.404} C_VEL
LIN {X 0,Y 285.574,Z 366.8,A -85,B 0,C 180,E1 -18363.807,E2 -18363.807} C_VEL
LIN {X 0,Y 285.602,Z 361.072,A -85,B 0,C 180,E1 -18364.091,E2 -18364.091} C_VEL
LIN {X 0,Y 285.965,Z 354.497,A -85,B 0,C 180,E1 -18364.353,E2 -18364.353} C_VEL
LIN {X 0,Y 281.72,Z 345.537,A -85,B 0,C 180,E1 -18365.767,E2 -18365.767} C_VEL
LIN {X 0,Y 276.547,Z 337.045,A -85,B 0,C 180,E1 -18367.554,E2 -18367.554} C_VEL
LIN {X 0,Y 271.676,Z 329.27,A -85,B 0,C 180,E1 -18369.442,E2 -18369.442} C_VEL
LIN {X 0,Y 267.332,Z 323.63,A -85,B 0,C 180,E1 -18371.24,E2 -18371.24} C_VEL
LIN {X 0,Y 263.079,Z 318.394,A -85,B 0,C 180,E1 -18373.224,E2 -18373.224} C_VEL
LIN {X 0,Y 260.348,Z 315.057,A -85,B 0,C 180,E1 -18374.695,E2 -18374.695} C_VEL
LIN {X 0,Y 258.103,Z 312.571,A -85,B 0,C 180,E1 -18375.995,E2 -18375.995} C_VEL
LIN {X 0,Y 256.935,Z 311.032,A -85,B 0,C 180,E1 -18376.819,E2 -18376.819} C_VEL
LIN {X 0,Y 256.102,Z 308.576,A -85,B 0,C 180,E1 -18379.853,E2 -18379.853} C_VEL
LIN {X 0,Y 256.137,Z 308.575,A -85,B 0,C 180,E1 -18385.132,E2 -18385.132} C_VEL
LIN {X 0,Y 256.083,Z 308.579,A -85,B 0,C 180,E1 -18388.588,E2 -18388.588} C_VEL
LIN {X 0,Y 256.045,Z 308.583,A -85,B 0,C 180,E1 -18391.705,E2 -18391.705} C_VEL
LIN {X 0,Y 256.115,Z 308.679,A -85,B 0,C 180,E1 -18395.913,E2 -18395.913} C_VEL
LIN {X 0,Y 257.595,Z 312.432,A -85,B 0,C 180,E1 -18400.199,E2 -18400.199} C_VEL
LIN {X 0,Y 258.795,Z 315.508,A -85,B 0,C 180,E1 -18402.852,E2 -18402.852} C_VEL
LIN {X 0,Y 260.998,Z 321.672,A -85,B 0,C 180,E1 -18407.055,E2 -18407.055} C_VEL
LIN {X 0,Y 261.499,Z 322.769,A -85,B 0,C 180,E1 -18407.516,E2 -18407.516} C_VEL
LIN {X 0,Y 266.16,Z 329.987,A -85,B 0,C 180,E1 -18409.853,E2 -18409.853} C_VEL
LIN {X 0,Y 270.345,Z 337.033,A -85,B 0,C 180,E1 -18411.703,E2 -18411.703} C_VEL
LIN {X 0,Y 273.386,Z 342.688,A -85,B 0,C 180,E1 -18412.962,E2 -18412.962} C_VEL
LIN {X 0,Y 276.201,Z 348.153,A -85,B 0,C 180,E1 -18414.039,E2 -18414.039} C_VEL
LIN {X 0,Y 280.584,Z 358.104,A -85,B 0,C 180,E1 -18415.691,E2 -18415.691} C_VEL
LIN {X 0,Y 281.426,Z 361.045,A -85,B 0,C 180,E1 -18416.035,E2 -18416.035} C_VEL
LIN {X 0,Y 283.268,Z 376.433,A -85,B 0,C 180,E1 -18417.233,E2 -18417.233} C_VEL
LIN {X 0,Y 284.076,Z 387.143,A -85,B 0,C 180,E1 -18417.942,E2 -18417.942} C_VEL
LIN {X 0,Y 280.108,Z 438.415,A -85,B 0,C 180,E1 -18419.719,E2 -18419.719} C_VEL
LIN {X 0,Y 278.346,Z 451.57,A -85,B 0,C 180,E1 -18420.406,E2 -18420.406} C_VEL
LIN {X 0,Y 276.084,Z 463.8,A -85,B 0,C 180,E1 -18421.289,E2 -18421.289} C_VEL
LIN {X 0,Y 273.473,Z 475.741,A -85,B 0,C 180,E1 -18422.452,E2 -18422.452} C_VEL
LIN {X 0,Y 270.689,Z 486.702,A -85,B 0,C 180,E1 -18423.814,E2 -18423.814} C_VEL
LIN {X 0,Y 267.558,Z 497.795,A -85,B 0,C 180,E1 -18425.567,E2 -18425.567} C_VEL
LIN {X 0,Y 264.834,Z 506.919,A -85,B 0,C 180,E1 -18427.374,E2 -18427.374} C_VEL
LIN {X 0,Y 261.907,Z 515.934,A -85,B 0,C 180,E1 -18429.588,E2 -18429.588} C_VEL
LIN {X 0,Y 259.546,Z 523.234,A -85,B 0,C 180,E1 -18431.861,E2 -18431.861} C_VEL
LIN {X 0,Y 257.679,Z 529.136,A -85,B 0,C 180,E1 -18434.177,E2 -18434.177} C_VEL
LIN {X 0,Y 256.023,Z 533.892,A -85,B 0,C 180,E1 -18436.511,E2 -18436.511} C_VEL
LIN {X 0,Y 255.008,Z 537.562,A -85,B 0,C 180,E1 -18438.881,E2 -18438.881} C_VEL
LIN {X 0,Y 254.558,Z 539.433,A -85,B 0,C 180,E1 -18440.468,E2 -18440.468} C_VEL
LIN {X 0,Y 254.148,Z 541.959,A -85,B 0,C 180,E1 -18443.653,E2 -18443.653} C_VEL
LIN {X 0,Y 254.066,Z 542.586,A -85,B 0,C 180,E1 -18445.243,E2 -18445.243} C_VEL
LIN {X 0,Y 254.178,Z 542.795,A -85,B 0,C 180,E1 -18446.833,E2 -18446.833} C_VEL
LIN {X 0,Y 254.206,Z 542.59,A -85,B 0,C 180,E1 -18448.418,E2 -18448.418} C_VEL
LIN {X 0,Y 254.413,Z 541.984,A -85,B 0,C 180,E1 -18450.003,E2 -18450.003} C_VEL
LIN {X 0,Y 254.286,Z 540.882,A -85,B 0,C 180,E1 -18451.586,E2 -18451.586} C_VEL
LIN {X 0,Y 254.301,Z 538.398,A -85,B 0,C 180,E1 -18453.964,E2 -18453.964} C_VEL
LIN {X 0,Y 254.362,Z 534.802,A -85,B 0,C 180,E1 -18456.347,E2 -18456.347} C_VEL
LIN {X 0,Y 254.49,Z 529.984,A -85,B 0,C 180,E1 -18458.738,E2 -18458.738} C_VEL
LIN {X 0,Y 254.93,Z 523.824,A -85,B 0,C 180,E1 -18461.128,E2 -18461.128} C_VEL
LIN {X 0,Y 255.768,Z 516.119,A -85,B 0,C 180,E1 -18463.508,E2 -18463.508} C_VEL
LIN {X 0,Y 256.718,Z 508.218,A -85,B 0,C 180,E1 -18465.482,E2 -18465.482} C_VEL
LIN {X 0,Y 257.953,Z 498.096,A -85,B 0,C 180,E1 -18467.523,E2 -18467.523} C_VEL
LIN {X 0,Y 259.295,Z 487.864,A -85,B 0,C 180,E1 -18469.187,E2 -18469.187} C_VEL
LIN {X 0,Y 260.705,Z 475.991,A -85,B 0,C 180,E1 -18470.722,E2 -18470.722} C_VEL
LIN {X 0,Y 262.09,Z 463.577,A -85,B 0,C 180,E1 -18471.947,E2 -18471.947} C_VEL
LIN {X 0,Y 263.173,Z 450.812,A -85,B 0,C 180,E1 -18472.886,E2 -18472.886} C_VEL
LIN {X 0,Y 263.973,Z 437.556,A -85,B 0,C 180,E1 -18473.538,E2 -18473.538} C_VEL
LIN {X 0,Y 265.998,Z 381.968,A -85,B 0,C 180,E1 -18475.425,E2 -18475.425} C_VEL
LIN {X 0,Y 260.608,Z 331.697,A -85,B 0,C 180,E1 -18477.678,E2 -18477.678} C_VEL
LIN {X 0,Y 259.478,Z 324.773,A -85,B 0,C 180,E1 -18479.918,E2 -18479.918} C_VEL
LIN {X 0,Y 256.94,Z 312.42,A -85,B 0,C 180,E1 -18484.105,E2 -18484.105} C_VEL
LIN {X 0,Y 256.145,Z 308.577,A -85,B 0,C 180,E1 -18485.483,E2 -18485.483} C_VEL
LIN {X 0,Y 256.025,Z 308.591,A -85,B 0,C 180,E1 -18489.77,E2 -18489.77} C_VEL
LIN {X 0,Y 256.017,Z 308.593,A -85,B 0,C 180,E1 -18493.335,E2 -18493.335} C_VEL
LIN {X 0,Y 256.025,Z 308.59,A -85,B 0,C 180,E1 -18497.828,E2 -18497.828} C_VEL
LIN {X 0,Y 256.057,Z 308.591,A -85,B 0,C 180,E1 -18500.854,E2 -18500.854} C_VEL
LIN {X 0,Y 256.07,Z 308.588,A -85,B 0,C 180,E1 -18504.804,E2 -18504.804} C_VEL
LIN {X 0,Y 256.068,Z 308.587,A -85,B 0,C 180,E1 -18508.568,E2 -18508.568} C_VEL
LIN {X 0,Y 256.083,Z 308.584,A -85,B 0,C 180,E1 -18512.189,E2 -18512.189} C_VEL
LIN {X 0,Y 256.12,Z 308.579,A -85,B 0,C 180,E1 -18515.694,E2 -18515.694} C_VEL
LIN {X 0,Y 256.11,Z 308.583,A -85,B 0,C 180,E1 -18519.099,E2 -18519.099} C_VEL
LIN {X 0,Y 256.214,Z 308.566,A -85,B 0,C 180,E1 -18524.079,E2 -18524.079} C_VEL
LIN {X 0,Y 256.263,Z 308.563,A -85,B 0,C 180,E1 -18528.931,E2 -18528.931} C_VEL
LIN {X 0,Y 256.493,Z 308.532,A -85,B 0,C 180,E1 -18532.125,E2 -18532.125} C_VEL
LIN {X 0,Y 256.47,Z 308.536,A -85,B 0,C 180,E1 -18536.858,E2 -18536.858} C_VEL
LIN {X 0,Y 256.724,Z 308.504,A -85,B 0,C 180,E1 -18539.999,E2 -18539.999} C_VEL
LIN {X 0,Y 256.469,Z 308.535,A -85,B 0,C 180,E1 -18543.141,E2 -18543.141} C_VEL
LIN {X 0,Y 256.49,Z 308.535,A -85,B 0,C 180,E1 -18547.874,E2 -18547.874} C_VEL
LIN {X 0,Y 256.241,Z 308.563,A -85,B 0,C 180,E1 -18552.674,E2 -18552.674} C_VEL
LIN {X 0,Y 256.199,Z 308.57,A -85,B 0,C 180,E1 -18556.248,E2 -18556.248} C_VEL
LIN {X 0,Y 256.107,Z 308.58,A -85,B 0,C 180,E1 -18561.098,E2 -18561.098} C_VEL
LIN {X 0,Y 256.157,Z 308.575,A -85,B 0,C 180,E1 -18565.129,E2 -18565.129} C_VEL
LIN {X 0,Y 256.091,Z 308.584,A -85,B 0,C 180,E1 -18569.602,E2 -18569.602} C_VEL
LIN {X 0,Y 256.056,Z 308.588,A -85,B 0,C 180,E1 -18573.293,E2 -18573.293} C_VEL
LIN {X 0,Y 256.11,Z 308.579,A -85,B 0,C 180,E1 -18577.273,E2 -18577.273} C_VEL
LIN {X 0,Y 256.065,Z 308.588,A -85,B 0,C 180,E1 -18582.182,E2 -18582.182} C_VEL
LIN {X 0,Y 256.091,Z 308.583,A -85,B 0,C 180,E1 -18586.681,E2 -18586.681} C_VEL
LIN {X 0,Y 256.102,Z 308.581,A -85,B 0,C 180,E1 -18590.865,E2 -18590.865} C_VEL
LIN {X 0,Y 256.116,Z 308.58,A -85,B 0,C 180,E1 -18594.814,E2 -18594.814} C_VEL
LIN {X 0,Y 256.087,Z 308.584,A -85,B 0,C 180,E1 -18598.572,E2 -18598.572} C_VEL
LIN {X 0,Y 256.134,Z 308.579,A -85,B 0,C 180,E1 -18602.196,E2 -18602.196} C_VEL
LIN {X 0,Y 256.165,Z 308.574,A -85,B 0,C 180,E1 -18605.699,E2 -18605.699} C_VEL
LIN {X 0,Y 256.167,Z 308.571,A -85,B 0,C 180,E1 -18609.104,E2 -18609.104} C_VEL
LIN {X 0,Y 256.298,Z 308.559,A -85,B 0,C 180,E1 -18614.084,E2 -18614.084} C_VEL
LIN {X 0,Y 256.308,Z 308.556,A -85,B 0,C 180,E1 -18618.933,E2 -18618.933} C_VEL
LIN {X 0,Y 256.538,Z 308.529,A -85,B 0,C 180,E1 -18622.125,E2 -18622.125} C_VEL
LIN {X 0,Y 256.712,Z 308.507,A -85,B 0,C 180,E1 -18628.429,E2 -18628.429} C_VEL
LIN {X 0,Y 256.712,Z 308.505,A -85,B 0,C 180,E1 -18631.566,E2 -18631.566} C_VEL
LIN {X 0,Y 256.535,Z 308.528,A -85,B 0,C 180,E1 -18637.87,E2 -18637.87} C_VEL
LIN {X 0,Y 256.305,Z 308.558,A -85,B 0,C 180,E1 -18641.063,E2 -18641.063} C_VEL
LIN {X 0,Y 256.292,Z 308.556,A -85,B 0,C 180,E1 -18645.911,E2 -18645.911} C_VEL
LIN {X 0,Y 256.222,Z 308.571,A -85,B 0,C 180,E1 -18650.885,E2 -18650.885} C_VEL
LIN {X 0,Y 256.177,Z 308.575,A -85,B 0,C 180,E1 -18655.135,E2 -18655.135} C_VEL
LIN {X 0,Y 256.099,Z 308.583,A -85,B 0,C 180,E1 -18659.595,E2 -18659.595} C_VEL
LIN {X 0,Y 256.132,Z 308.661,A -85,B 0,C 180,E1 -18664.344,E2 -18664.344} C_VEL
LIN {X 0,Y 266.076,Z 335.715,A -85,B 0,C 180,E1 -18666.082,E2 -18666.082} C_VEL
LIN {X 0,Y 267.048,Z 338.659,A -85,B 0,C 180,E1 -18666.254,E2 -18666.254} C_VEL
LIN {X 0,Y 264.128,Z 411.88,A -85,B 0,C 180,E1 -18668.745,E2 -18668.745} C_VEL
LIN {X 0,Y 263.482,Z 425.479,A -85,B 0,C 180,E1 -18669.521,E2 -18669.521} C_VEL
LIN {X 0,Y 262.444,Z 438.259,A -85,B 0,C 180,E1 -18670.55,E2 -18670.55} C_VEL
LIN {X 0,Y 261.308,Z 450.411,A -85,B 0,C 180,E1 -18671.858,E2 -18671.858} C_VEL
LIN {X 0,Y 259.982,Z 461.667,A -85,B 0,C 180,E1 -18673.39,E2 -18673.39} C_VEL
LIN {X 0,Y 258.676,Z 472.893,A -85,B 0,C 180,E1 -18675.333,E2 -18675.333} C_VEL
LIN {X 0,Y 257.383,Z 482.897,A -85,B 0,C 180,E1 -18677.488,E2 -18677.488} C_VEL
LIN {X 0,Y 256.352,Z 490.793,A -85,B 0,C 180,E1 -18679.606,E2 -18679.606} C_VEL
LIN {X 0,Y 255.416,Z 498.672,A -85,B 0,C 180,E1 -18682.25,E2 -18682.25} C_VEL
LIN {X 0,Y 254.824,Z 504.198,A -85,B 0,C 180,E1 -18684.608,E2 -18684.608} C_VEL
LIN {X 0,Y 254.533,Z 507.682,A -85,B 0,C 180,E1 -18686.481,E2 -18686.481} C_VEL
LIN {X 0,Y 254.158,Z 511.303,A -85,B 0,C 180,E1 -18688.991,E2 -18688.991} C_VEL
LIN {X 0,Y 254.002,Z 514.123,A -85,B 0,C 180,E1 -18691.942,E2 -18691.942} C_VEL
LIN {X 0,Y 254.104,Z 515.075,A -85,B 0,C 180,E1 -18693.736,E2 -18693.736} C_VEL
LIN {X 0,Y 254.413,Z 515.564,A -85,B 0,C 180,E1 -18695.709,E2 -18695.709} C_VEL
LIN {X 0,Y 254.738,Z 515.461,A -85,B 0,C 180,E1 -18697.28,E2 -18697.28} C_VEL
LIN {X 0,Y 255.388,Z 514.76,A -85,B 0,C 180,E1 -18699.31,E2 -18699.31} C_VEL
LIN {X 0,Y 255.952,Z 513.829,A -85,B 0,C 180,E1 -18700.763,E2 -18700.763} C_VEL
LIN {X 0,Y 257.082,Z 511.589,A -85,B 0,C 180,E1 -18703.073,E2 -18703.073} C_VEL
LIN {X 0,Y 258.867,Z 507.536,A -85,B 0,C 180,E1 -18705.858,E2 -18705.858} C_VEL
LIN {X 0,Y 260.907,Z 502.55,A -85,B 0,C 180,E1 -18708.345,E2 -18708.345} C_VEL
LIN {X 0,Y 263.395,Z 496.126,A -85,B 0,C 180,E1 -18710.788,E2 -18710.788} C_VEL
LIN {X 0,Y 265.716,Z 489.501,A -85,B 0,C 180,E1 -18712.783,E2 -18712.783} C_VEL
LIN {X 0,Y 268.572,Z 480.67,A -85,B 0,C 180,E1 -18714.898,E2 -18714.898} C_VEL
LIN {X 0,Y 271.587,Z 470.45,A -85,B 0,C 180,E1 -18716.848,E2 -18716.848} C_VEL
LIN {X 0,Y 274.16,Z 460.266,A -85,B 0,C 180,E1 -18718.4,E2 -18718.4} C_VEL
LIN {X 0,Y 276.724,Z 448.301,A -85,B 0,C 180,E1 -18719.828,E2 -18719.828} C_VEL
LIN {X 0,Y 278.928,Z 435.559,A -85,B 0,C 180,E1 -18720.993,E2 -18720.993} C_VEL
LIN {X 0,Y 280.651,Z 422.235,A -85,B 0,C 180,E1 -18721.872,E2 -18721.872} C_VEL
LIN {X 0,Y 281.831,Z 409.242,A -85,B 0,C 180,E1 -18722.45,E2 -18722.45} C_VEL
LIN {X 0,Y 285.602,Z 361.072,A -85,B 0,C 180,E1 -18724.091,E2 -18724.091} C_VEL
LIN {X 0,Y 285.242,Z 358.202,A -85,B 0,C 180,E1 -18724.319,E2 -18724.319} C_VEL
LIN {X 0,Y 283.765,Z 355.475,A -85,B 0,C 180,E1 -18724.787,E2 -18724.787} C_VEL
LIN {X 0,Y 282.113,Z 353.743,A -85,B 0,C 180,E1 -18725.252,E2 -18725.252} C_VEL
LIN {X 0,Y 277.57,Z 349.741,A -85,B 0,C 180,E1 -18726.55,E2 -18726.55} C_VEL
LIN {X 0,Y 276.385,Z 347.949,A -85,B 0,C 180,E1 -18726.951,E2 -18726.951} C_VEL
LIN {X 0,Y 269.758,Z 337.061,A -85,B 0,C 180,E1 -18729.503,E2 -18729.503} C_VEL
LIN {X 0,Y 265.283,Z 330.493,A -85,B 0,C 180,E1 -18731.456,E2 -18731.456} C_VEL
LIN {X 0,Y 260.696,Z 324.732,A -85,B 0,C 180,E1 -18733.682,E2 -18733.682} C_VEL
LIN {X 0,Y 257.667,Z 321.029,A -85,B 0,C 180,E1 -18735.373,E2 -18735.373} C_VEL
LIN {X 0,Y 255.637,Z 318.706,A -85,B 0,C 180,E1 -18736.642,E2 -18736.642} C_VEL
LIN {X 0,Y 254.055,Z 317.006,A -85,B 0,C 180,E1 -18737.717,E2 -18737.717} C_VEL
LIN {X 0,Y 250.305,Z 312.674,A -85,B 0,C 180,E1 -18740.88,E2 -18740.88} C_VEL
LIN {X 0,Y 249.453,Z 311.009,A -85,B 0,C 180,E1 -18745.655,E2 -18745.655} C_VEL
LIN {X 0,Y 249.357,Z 310.947,A -85,B 0,C 180,E1 -18749.122,E2 -18749.122} C_VEL
LIN {X 0,Y 250.126,Z 312.442,A -85,B 0,C 180,E1 -18754.192,E2 -18754.192} C_VEL
LIN {X 0,Y 250.736,Z 313.41,A -85,B 0,C 180,E1 -18756.06,E2 -18756.06} C_VEL
LIN {X 0,Y 251.977,Z 316.676,A -85,B 0,C 180,E1 -18759.905,E2 -18759.905} C_VEL
LIN {X 0,Y 253.552,Z 320.909,A -85,B 0,C 180,E1 -18763.461,E2 -18763.461} C_VEL
LIN {X 0,Y 259.063,Z 329.102,A -85,B 0,C 180,E1 -18767.024,E2 -18767.024} C_VEL
LIN {X 0,Y 263.227,Z 335.803,A -85,B 0,C 180,E1 -18769.234,E2 -18769.234} C_VEL
LIN {X 0,Y 267.135,Z 342.714,A -85,B 0,C 180,E1 -18771.085,E2 -18771.085} C_VEL
LIN {X 0,Y 269.814,Z 347.798,A -85,B 0,C 180,E1 -18772.246,E2 -18772.246} C_VEL
LIN {X 0,Y 272.996,Z 354.338,A -85,B 0,C 180,E1 -18773.57,E2 -18773.57} C_VEL
LIN {X 0,Y 276.737,Z 363.397,A -85,B 0,C 180,E1 -18775.055,E2 -18775.055} C_VEL
LIN {X 0,Y 278.299,Z 377.895,A -85,B 0,C 180,E1 -18776.232,E2 -18776.232} C_VEL
LIN {X 0,Y 279.051,Z 388.344,A -85,B 0,C 180,E1 -18776.946,E2 -18776.946} C_VEL
LIN {X 0,Y 274.975,Z 437.48,A -85,B 0,C 180,E1 -18778.677,E2 -18778.677} C_VEL
LIN {X 0,Y 272.966,Z 451.748,A -85,B 0,C 180,E1 -18779.442,E2 -18779.442} C_VEL
LIN {X 0,Y 270.407,Z 464.63,A -85,B 0,C 180,E1 -18780.414,E2 -18780.414} C_VEL
LIN {X 0,Y 267.684,Z 476.343,A -85,B 0,C 180,E1 -18781.59,E2 -18781.59} C_VEL
LIN {X 0,Y 264.783,Z 487.129,A -85,B 0,C 180,E1 -18782.97,E2 -18782.97} C_VEL
LIN {X 0,Y 261.827,Z 497.029,A -85,B 0,C 180,E1 -18784.571,E2 -18784.571} C_VEL
LIN {X 0,Y 258.834,Z 506.144,A -85,B 0,C 180,E1 -18786.396,E2 -18786.396} C_VEL
LIN {X 0,Y 255.749,Z 515.16,A -85,B 0,C 180,E1 -18788.652,E2 -18788.652} C_VEL
LIN {X 0,Y 253.16,Z 522.578,A -85,B 0,C 180,E1 -18790.981,E2 -18790.981} C_VEL
LIN {X 0,Y 250.863,Z 529.354,A -85,B 0,C 180,E1 -18793.735,E2 -18793.735} C_VEL
LIN {X 0,Y 249.103,Z 533.936,A -85,B 0,C 180,E1 -18796.129,E2 -18796.129} C_VEL
LIN {X 0,Y 248.021,Z 537.461,A -85,B 0,C 180,E1 -18798.563,E2 -18798.563} C_VEL
LIN {X 0,Y 247.536,Z 539.275,A -85,B 0,C 180,E1 -18800.195,E2 -18800.195} C_VEL
LIN {X 0,Y 247.186,Z 540.679,A -85,B 0,C 180,E1 -18801.831,E2 -18801.831} C_VEL
LIN {X 0,Y 246.991,Z 542.141,A -85,B 0,C 180,E1 -18804.821,E2 -18804.821} C_VEL
LIN {X 0,Y 247.105,Z 542.352,A -85,B 0,C 180,E1 -18806.742,E2 -18806.742} C_VEL
LIN {X 0,Y 247.13,Z 542.094,A -85,B 0,C 180,E1 -18808.373,E2 -18808.373} C_VEL
LIN {X 0,Y 247.33,Z 541.406,A -85,B 0,C 180,E1 -18810.003,E2 -18810.003} C_VEL
LIN {X 0,Y 247.207,Z 540.226,A -85,B 0,C 180,E1 -18811.632,E2 -18811.632} C_VEL
LIN {X 0,Y 247.247,Z 537.628,A -85,B 0,C 180,E1 -18814.077,E2 -18814.077} C_VEL
LIN {X 0,Y 247.274,Z 533.901,A -85,B 0,C 180,E1 -18816.53,E2 -18816.53} C_VEL
LIN {X 0,Y 247.439,Z 528.947,A -85,B 0,C 180,E1 -18818.989,E2 -18818.989} C_VEL
LIN {X 0,Y 247.931,Z 522.637,A -85,B 0,C 180,E1 -18821.446,E2 -18821.446} C_VEL
LIN {X 0,Y 248.835,Z 514.724,A -85,B 0,C 180,E1 -18823.892,E2 -18823.892} C_VEL
LIN {X 0,Y 250.077,Z 504.757,A -85,B 0,C 180,E1 -18826.323,E2 -18826.323} C_VEL
LIN {X 0,Y 251.273,Z 495.562,A -85,B 0,C 180,E1 -18828.13,E2 -18828.13} C_VEL
LIN {X 0,Y 252.765,Z 484.212,A -85,B 0,C 180,E1 -18829.914,E2 -18829.914} C_VEL
LIN {X 0,Y 254.013,Z 473.177,A -85,B 0,C 180,E1 -18831.294,E2 -18831.294} C_VEL
LIN {X 0,Y 255.349,Z 461.24,A -85,B 0,C 180,E1 -18832.451,E2 -18832.451} C_VEL
LIN {X 0,Y 256.485,Z 447.518,A -85,B 0,C 180,E1 -18833.411,E2 -18833.411} C_VEL
LIN {X 0,Y 257.16,Z 435.296,A -85,B 0,C 180,E1 -18833.987,E2 -18833.987} C_VEL
LIN {X 0,Y 259.106,Z 381.94,A -85,B 0,C 180,E1 -18835.856,E2 -18835.856} C_VEL
